KUKA KRL program: MyProgram_267().src

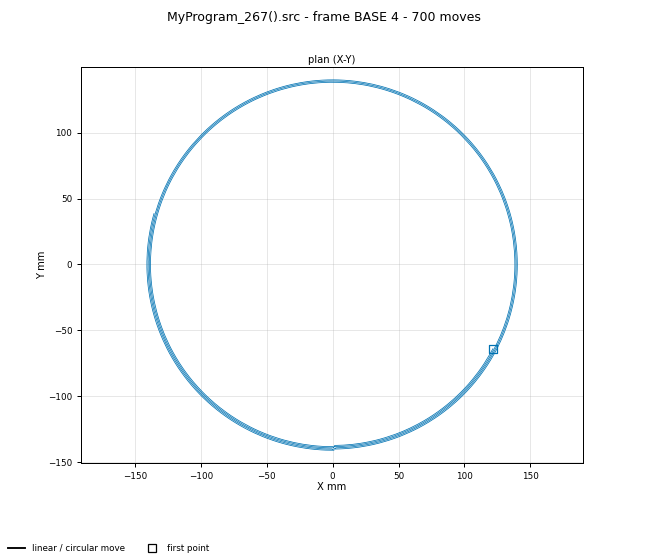
[picture p0: tool path of MyProgram_267().src in frame BASE 4, 700 of 700 moves have a stored position in this frame; points joined in program order, loops and branches not executed]
&ACCESS RVP
&REL 1
&PARAM TEMPLATE = C:\KRC\Roboter\Template\vorgabe
&PARAM EDITMASK = *
DEF MyProgram_267()
; ---- Setting reference (Base) ----
$BASE = BASE_DATA[4]

; --------------------------
; ---- Setting tool (TCP) ----
$TOOL = TOOL_DATA[3]
; --------------------------

$VEL.CP = VEL_APROX_PRINT
Startdeposition()
$VEL.CP = VEL_PRINT
LIN {X 121.5223,Y -63.9531,Z 169,A -26.4132,B 9.7444,C 0.283,E1 9.8897,E2 477.634} C_DIS
LIN {X 119.4927,Y -67.6748,Z 169,A -28.3857,B 9.744,C 0.2925,E1 9.8869,E2 479.6342} C_DIS
LIN {X 114.8477,Y -75.2879,Z 169,A -31.797,B 9.744,C 0.2945,E1 9.882,E2 483.0104} C_DIS
LIN {X 112.9327,Y -78.1315,Z 169,A -33.3387,B 9.7438,C 0.3007,E1 9.8795,E2 484.5678} C_DIS
LIN {X 110.5893,Y -81.4139,Z 169,A -34.9698,B 9.7438,C 0.3035,E1 9.8769,E2 486.1941} C_DIS
LIN {X 107.7784,Y -85.1007,Z 169,A -36.6917,B 9.7438,C 0.303,E1 9.874,E2 487.8912} C_DIS
LIN {X 105.9489,Y -87.3676,Z 169,A -38.1579,B 9.7434,C 0.3119,E1 9.8713,E2 489.3904} C_DIS
LIN {X 103.0991,Y -90.7131,Z 169,A -40.1493,B 9.7432,C 0.3198,E1 9.8676,E2 491.4037} C_DIS
LIN {X 100.8727,Y -93.1825,Z 169,A -41.7921,B 9.7429,C 0.3289,E1 9.8645,E2 493.08} C_DIS
LIN {X 97.5521,Y -96.653,Z 169,A -43.3158,B 9.7431,C 0.3219,E1 9.8616,E2 494.5453} C_DIS
LIN {X 92.7016,Y -101.3149,Z 169,A -46.0443,B 9.743,C 0.3259,E1 9.8561,E2 497.2667} C_DIS
LIN {X 87.8927,Y -105.5141,Z 169,A -48.4523,B 9.743,C 0.3252,E1 9.8511,E2 499.6449} C_DIS
LIN {X 83.878,Y -108.7326,Z 169,A -51.2584,B 9.7423,C 0.3447,E1 9.8447,E2 502.5365} C_DIS
LIN {X 80.2624,Y -111.4281,Z 169,A -52.6799,B 9.7426,C 0.3374,E1 9.8416,E2 503.9017} C_DIS
LIN {X 76.6421,Y -113.9489,Z 169,A -54.4958,B 9.7426,C 0.34,E1 9.8374,E2 505.7163} C_DIS
LIN {X 73.1697,Y -116.2085,Z 169,A -56.1855,B 9.7424,C 0.342,E1 9.8335,E2 507.4026} C_DIS
LIN {X 69.7328,Y -118.3029,Z 169,A -57.7924,B 9.7424,C 0.343,E1 9.8296,E2 509.0019} C_DIS
LIN {X 64.6366,Y -121.163,Z 169,A -60.2336,B 9.7423,C 0.3468,E1 9.8237,E2 511.4457} C_DIS
LIN {X 61.9846,Y -122.5384,Z 169,A -61.5098,B 9.7422,C 0.3493,E1 9.8205,E2 512.7266} C_DIS
LIN {X 58.8364,Y -124.081,Z 169,A -62.8714,B 9.7422,C 0.349,E1 9.8171,E2 514.0767} C_DIS
LIN {X 54.0796,Y -126.227,Z 169,A -65.0052,B 9.7422,C 0.3508,E1 9.8117,E2 516.2068} C_DIS
LIN {X 51.4311,Y -127.3284,Z 169,A -66.2612,B 9.742,C 0.3536,E1 9.8084,E2 517.4712} C_DIS
LIN {X 47.3484,Y -128.9049,Z 169,A -68.3007,B 9.7418,C 0.3606,E1 9.803,E2 519.5393} C_DIS
LIN {X 42.0304,Y -130.7333,Z 169,A -70.1991,B 9.7421,C 0.3529,E1 9.7981,E2 521.3826} C_DIS
LIN {X 40.0355,Y -131.3578,Z 169,A -71.2939,B 9.7418,C 0.3588,E1 9.7951,E2 522.5064} C_DIS
LIN {X 36.2701,Y -132.449,Z 169,A -72.8975,B 9.7418,C 0.3596,E1 9.7908,E2 524.1071} C_DIS
LIN {X 32.8798,Y -133.331,Z 169,A -74.3211,B 9.7418,C 0.3599,E1 9.787,E2 525.5269} C_DIS
LIN {X 28.4405,Y -134.3472,Z 169,A -76.2879,B 9.7417,C 0.3629,E1 9.7816,E2 527.5034} C_DIS
LIN {X 25.1446,Y -135.0034,Z 169,A -77.8597,B 9.7415,C 0.3675,E1 9.7772,E2 529.0976} C_DIS
LIN {X 21.1222,Y -135.6894,Z 169,A -79.3371,B 9.7417,C 0.3636,E1 9.7732,E2 530.5475} C_DIS
LIN {X 15.2674,Y -136.4735,Z 169,A -81.7848,B 9.7417,C 0.3645,E1 9.7664,E2 532.9947} C_DIS
LIN {X 8.3393,Y -137.0702,Z 169,A -84.7346,B 9.7416,C 0.3666,E1 9.7582,E2 535.9522} C_DIS
LIN {X 1.6144,Y -137.3159,Z 169,A -87.597,B 9.7415,C 0.3684,E1 9.7502,E2 538.8231} C_DIS
LIN {X 1.6144,Y -137.3159,Z 169,A -87.597,B 9.7415,C 0.3684,E1 9.7502,E2 538.8231} C_DIS
Enddeposition()
LIN {X 1.0035,Y -138.2302,Z 169,A -87.3337,B 9.7081,C 0.3639,E1 9.7175,E2 538.5378} C_DIS
Startdeposition()
$VEL.CP = VEL_PRINT
LIN {X 3.6243,Y -138.1887,Z 169,A -85.9275,B 9.7084,C 0.3567,E1 9.7215,E2 537.0898} C_DIS
LIN {X 8.1585,Y -137.9955,Z 169,A -84.3267,B 9.7082,C 0.3624,E1 9.7259,E2 535.5242} C_DIS
LIN {X 12.5987,Y -137.662,Z 169,A -82.2235,B 9.7084,C 0.3561,E1 9.7318,E2 533.3868} C_DIS
LIN {X 15.47,Y -137.3693,Z 169,A -80.2721,B 9.709,C 0.3386,E1 9.7375,E2 531.3363} C_DIS
LIN {X 21.6232,Y -136.5351,Z 169,A -78.7263,B 9.7082,C 0.3603,E1 9.7414,E2 529.9229} C_DIS
LIN {X 27.0044,Y -135.5737,Z 169,A -76.2156,B 9.7085,C 0.3533,E1 9.7484,E2 527.3791} C_DIS
LIN {X 31.4408,Y -134.6145,Z 169,A -73.9888,B 9.7088,C 0.344,E1 9.7546,E2 525.1061} C_DIS
LIN {X 35.2299,Y -133.6717,Z 169,A -72.753,B 9.7086,C 0.3514,E1 9.7578,E2 523.9189} C_DIS
LIN {X 38.6757,Y -132.7152,Z 169,A -71.3127,B 9.7086,C 0.351,E1 9.7616,E2 522.483} C_DIS
LIN {X 42.1668,Y -131.6475,Z 169,A -69.2693,B 9.7091,C 0.3373,E1 9.7673,E2 520.3694} C_DIS
LIN {X 46.617,Y -130.1385,Z 169,A -68.083,B 9.7085,C 0.3527,E1 9.7702,E2 519.2806} C_DIS
LIN {X 51.6048,Y -128.2421,Z 169,A -65.7308,B 9.7087,C 0.3469,E1 9.7763,E2 516.9086} C_DIS
LIN {X 58.3851,Y -125.3013,Z 169,A -62.6142,B 9.7089,C 0.3418,E1 9.7843,E2 513.7827} C_DIS
LIN {X 62.2786,Y -123.4126,Z 169,A -60.8218,B 9.7089,C 0.3393,E1 9.7888,E2 511.989} C_DIS
LIN {X 65.0912,Y -121.9545,Z 169,A -59.5881,B 9.7089,C 0.3393,E1 9.7918,E2 510.7645} C_DIS
LIN {X 68.9115,Y -119.8373,Z 169,A -57.5572,B 9.7093,C 0.3313,E1 9.7968,E2 508.7033} C_DIS
LIN {X 73.8951,Y -116.8295,Z 169,A -55.2807,B 9.7093,C 0.3305,E1 9.8022,E2 506.4423} C_DIS
LIN {X 77.7185,Y -114.322,Z 169,A -53.6415,B 9.7092,C 0.3333,E1 9.8059,E2 504.8345} C_DIS
LIN {X 81.5319,Y -111.6347,Z 169,A -50.4812,B 9.7103,C 0.3005,E1 9.8135,E2 501.5122} C_DIS
LIN {X 87.6058,Y -106.9339,Z 169,A -47.584,B 9.7103,C 0.3013,E1 9.8196,E2 498.6497} C_DIS
LIN {X 92.3827,Y -102.8352,Z 169,A -45.9634,B 9.7096,C 0.3198,E1 9.8228,E2 497.1552} C_DIS
LIN {X 96.5302,Y -98.9528,Z 169,A -43.3774,B 9.71,C 0.3094,E1 9.8281,E2 494.537} C_DIS
LIN {X 102.34,Y -92.9307,Z 169,A -40.2491,B 9.71,C 0.31,E1 9.834,E2 491.4493} C_DIS
LIN {X 105.7678,Y -89.0102,Z 169,A -37.829,B 9.7103,C 0.2988,E1 9.8385,E2 488.9932} C_DIS
LIN {X 110.706,Y -82.7881,Z 169,A -34.445,B 9.7106,C 0.2888,E1 9.8443,E2 485.5939} C_DIS
LIN {X 113.6513,Y -78.6962,Z 169,A -32.5038,B 9.7106,C 0.2873,E1 9.8474,E2 483.6697} C_DIS
LIN {X 115.518,Y -75.929,Z 169,A -30.804,B 9.711,C 0.2761,E1 9.8501,E2 481.9274} C_DIS
LIN {X 117.7858,Y -72.361,Z 169,A -29.4472,B 9.7108,C 0.2813,E1 9.852,E2 480.62} C_DIS
LIN {X 119.8827,Y -68.8324,Z 169,A -27.7305,B 9.711,C 0.2766,E1 9.8544,E2 478.8995} C_DIS
LIN {X 121.9811,Y -65.0416,Z 169,A -25.9549,B 9.711,C 0.2724,E1 9.8568,E2 477.1247} C_DIS
LIN {X 124.1565,Y -60.7815,Z 169,A -23.1233,B 9.7118,C 0.2461,E1 9.8604,E2 474.1803} C_DIS
LIN {X 127.1987,Y -54.1312,Z 169,A -21.0317,B 9.7114,C 0.2612,E1 9.8626,E2 472.2079} C_DIS
LIN {X 129.7662,Y -47.6495,Z 169,A -18.1375,B 9.7116,C 0.2531,E1 9.8655,E2 469.3101} C_DIS
LIN {X 131.1674,Y -43.6372,Z 169,A -16.5544,B 9.7116,C 0.2526,E1 9.8669,E2 467.748} C_DIS
LIN {X 132.0304,Y -40.9555,Z 169,A -14.6508,B 9.7121,C 0.2311,E1 9.8686,E2 465.7479} C_DIS
LIN {X 133.6372,Y -35.3594,Z 169,A -12.9817,B 9.7119,C 0.2427,E1 9.8697,E2 464.1727} C_DIS
LIN {X 134.6403,Y -31.3276,Z 169,A -11.2449,B 9.7119,C 0.2374,E1 9.8709,E2 462.4322} C_DIS
LIN {X 136.0297,Y -24.5995,Z 169,A -8.547,B 9.7121,C 0.2329,E1 9.8723,E2 459.7506} C_DIS
LIN {X 137.2624,Y -16.3765,Z 169,A -5.3848,B 9.7121,C 0.23,E1 9.8736,E2 456.6214} C_DIS
LIN {X 137.5318,Y -13.94,Z 169,A -3.6442,B 9.7126,C 0.2091,E1 9.8741,E2 454.7869} C_DIS
LIN {X 137.9056,Y -9.5653,Z 169,A -2.3869,B 9.7124,C 0.2178,E1 9.8744,E2 453.6001} C_DIS
LIN {X 138.1517,Y -4.8579,Z 169,A -0.3244,B 9.7126,C 0.2094,E1 9.8746,E2 451.5217} C_DIS
LIN {X 138.2326,Y -1.1208,Z 169,A 1.7321,B 9.713,C 0.1923,E1 9.8746,E2 449.3985} C_DIS
LIN {X 138.1805,Y 3.9204,Z 169,A 3.8684,B 9.7131,C 0.185,E1 9.8745,E2 447.2541} C_DIS
LIN {X 137.9104,Y 9.4997,Z 169,A 5.533,B 9.7129,C 0.1944,E1 9.8742,E2 445.6712} C_DIS
LIN {X 137.1413,Y 17.3717,Z 169,A 8.5943,B 9.713,C 0.1903,E1 9.8733,E2 442.6347} C_DIS
LIN {X 136.3718,Y 22.6254,Z 169,A 10.9146,B 9.7132,C 0.1811,E1 9.8723,E2 440.2971} C_DIS
LIN {X 135.6149,Y 26.8018,Z 169,A 12.8909,B 9.7134,C 0.1707,E1 9.8713,E2 438.2917} C_DIS
LIN {X 134.9256,Y 30.0788,Z 169,A 14.0849,B 9.7134,C 0.1716,E1 9.8706,E2 437.1213} C_DIS
LIN {X 134.0282,Y 33.8467,Z 169,A 15.5369,B 9.7134,C 0.1708,E1 9.8696,E2 435.6875} C_DIS
LIN {X 133.1585,Y 37.1205,Z 169,A 16.9008,B 9.7134,C 0.1678,E1 9.8686,E2 434.3275} C_DIS
LIN {X 132.2106,Y 40.3666,Z 169,A 18.3307,B 9.7135,C 0.1632,E1 9.8675,E2 432.8929} C_DIS
LIN {X 131.1435,Y 43.7089,Z 169,A 19.7573,B 9.7135,C 0.1599,E1 9.8662,E2 431.4687} C_DIS
LIN {X 130.0245,Y 46.933,Z 169,A 21.422,B 9.7137,C 0.15,E1 9.8646,E2 429.771} C_DIS
LIN {X 128.8641,Y 50.0313,Z 169,A 22.6119,B 9.7137,C 0.1507,E1 9.8635,E2 428.6033} C_DIS
LIN {X 127.1009,Y 54.3573,Z 169,A 24.3261,B 9.7137,C 0.1509,E1 9.8617,E2 426.9159} C_DIS
LIN {X 125.6911,Y 57.5421,Z 169,A 25.6983,B 9.7137,C 0.1488,E1 9.8601,E2 425.5518} C_DIS
LIN {X 124.288,Y 60.5148,Z 169,A 27.2672,B 9.7139,C 0.1403,E1 9.8582,E2 423.9559} C_DIS
LIN {X 122.5937,Y 63.875,Z 169,A 28.7368,B 9.7139,C 0.1385,E1 9.8563,E2 422.4966} C_DIS
LIN {X 120.4568,Y 67.8217,Z 169,A 30.5977,B 9.7139,C 0.1338,E1 9.8538,E2 420.6345} C_DIS
LIN {X 117.4731,Y 72.8679,Z 169,A 33.0483,B 9.714,C 0.1273,E1 9.8503,E2 418.1799} C_DIS
LIN {X 115.0774,Y 76.5952,Z 169,A 34.8875,B 9.714,C 0.1228,E1 9.8474,E2 416.3394} C_DIS
LIN {X 112.2801,Y 80.6403,Z 169,A 36.8588,B 9.7141,C 0.1196,E1 9.8443,E2 414.3755} C_DIS
LIN {X 110.4497,Y 83.1294,Z 169,A 38.5654,B 9.7143,C 0.1065,E1 9.8413,E2 412.6141} C_DIS
LIN {X 107.5833,Y 86.8069,Z 169,A 40.1356,B 9.7143,C 0.1108,E1 9.8387,E2 411.0891} C_DIS
LIN {X 104.4049,Y 90.6056,Z 169,A 41.928,B 9.7143,C 0.1125,E1 9.8355,E2 409.3287} C_DIS
LIN {X 97.6535,Y 97.8442,Z 169,A 45.8298,B 9.7143,C 0.1087,E1 9.8281,E2 405.451} C_DIS
LIN {X 94.3854,Y 101.0003,Z 169,A 48.007,B 9.7143,C 0.0981,E1 9.8236,E2 403.2363} C_DIS
LIN {X 91.0289,Y 104.0355,Z 169,A 49.7708,B 9.7143,C 0.0971,E1 9.8199,E2 401.486} C_DIS
LIN {X 86.2559,Y 108.0258,Z 169,A 52.43,B 9.7144,C 0.0906,E1 9.8142,E2 398.816} C_DIS
LIN {X 82.0554,Y 111.2501,Z 169,A 55.1586,B 9.7146,C 0.0744,E1 9.8079,E2 396.0195} C_DIS
LIN {X 77.6146,Y 114.3924,Z 169,A 56.808,B 9.7145,C 0.0848,E1 9.8043,E2 394.4463} C_DIS
LIN {X 73.7755,Y 116.905,Z 169,A 58.6399,B 9.7145,C 0.0834,E1 9.8,E2 392.6229} C_DIS
LIN {X 70.2078,Y 119.082,Z 169,A 60.4141,B 9.7145,C 0.0799,E1 9.7957,E2 390.8433} C_DIS
LIN {X 66.413,Y 121.2394,Z 169,A 62.1811,B 9.7145,C 0.0784,E1 9.7914,E2 389.0814} C_DIS
LIN {X 58.9104,Y 125.0567,Z 169,A 65.5976,B 9.7145,C 0.0756,E1 9.7829,E2 385.6741} C_DIS
LIN {X 55.2301,Y 126.7236,Z 169,A 67.2877,B 9.7145,C 0.0733,E1 9.7786,E2 383.982} C_DIS
LIN {X 50.5322,Y 128.6694,Z 169,A 69.4095,B 9.7146,C 0.0708,E1 9.7731,E2 381.8586} C_DIS
LIN {X 47.1906,Y 129.9316,Z 169,A 70.8642,B 9.7146,C 0.0699,E1 9.7693,E2 380.4073} C_DIS
LIN {X 43.8069,Y 131.1109,Z 169,A 72.2508,B 9.7146,C 0.0707,E1 9.7657,E2 379.0331} C_DIS
LIN {X 40.5239,Y 132.1625,Z 169,A 73.7076,B 9.7146,C 0.0689,E1 9.7618,E2 377.5731} C_DIS
LIN {X 37.2525,Y 133.1216,Z 169,A 75.1127,B 9.7146,C 0.068,E1 9.758,E2 376.1693} C_DIS
LIN {X 33.8959,Y 134.0157,Z 169,A 77.457,B 9.7147,C 0.0472,E1 9.7514,E2 373.7115} C_DIS
LIN {X 27.4409,Y 135.4849,Z 169,A 79.3116,B 9.7147,C 0.0651,E1 9.7466,E2 371.9696} C_DIS
LIN {X 23.3469,Y 136.2514,Z 169,A 80.9226,B 9.7147,C 0.0667,E1 9.7422,E2 370.3735} C_DIS
LIN {X 16.9282,Y 137.1966,Z 169,A 83.5898,B 9.7147,C 0.0662,E1 9.7349,E2 367.7099} C_DIS
LIN {X 11.2415,Y 137.7787,Z 169,A 86.0643,B 9.7147,C 0.0634,E1 9.7279,E2 365.2233} C_DIS
LIN {X 4.1252,Y 138.1748,Z 169,A 89.0412,B 9.7147,C 0.0626,E1 9.7196,E2 362.2449} C_DIS
LIN {X -1.4773,Y 138.2301,Z 169,A 91.4614,B 9.7147,C 0.0606,E1 9.7128,E2 359.8137} C_DIS
LIN {X -4.6109,Y 138.1612,Z 169,A 93.452,B 9.7147,C 0.0462,E1 9.7071,E2 357.7371} C_DIS
LIN {X -10.677,Y 137.8244,Z 169,A 95.3517,B 9.7147,C 0.0598,E1 9.702,E2 355.9164} C_DIS
LIN {X -15.8973,Y 137.3196,Z 169,A 97.4052,B 9.7147,C 0.0631,E1 9.6963,E2 353.879} C_DIS
LIN {X -18.8245,Y 136.9502,Z 169,A 99.1396,B 9.7147,C 0.053,E1 9.6914,E2 352.0815} C_DIS
LIN {X -23.5939,Y 136.2096,Z 169,A 100.6893,B 9.7147,C 0.0634,E1 9.6872,E2 350.5895} C_DIS
LIN {X -28.7916,Y 135.2048,Z 169,A 102.7072,B 9.7147,C 0.0683,E1 9.6818,E2 348.5948} C_DIS
LIN {X -31.8808,Y 134.5103,Z 169,A 104.1791,B 9.7147,C 0.0659,E1 9.6777,E2 347.104} C_DIS
LIN {X -35.5184,Y 133.5948,Z 169,A 105.5905,B 9.7147,C 0.07,E1 9.6739,E2 345.7115} C_DIS
LIN {X -38.5661,Y 132.7473,Z 169,A 106.9576,B 9.7147,C 0.07,E1 9.6703,E2 344.3383} C_DIS
LIN {X -41.9093,Y 131.7298,Z 169,A 108.392,B 9.7147,C 0.0716,E1 9.6664,E2 342.9067} C_DIS
LIN {X -47.9387,Y 129.6579,Z 169,A 111.2253,B 9.7147,C 0.0704,E1 9.6589,E2 340.0518} C_DIS
LIN {X -51.8181,Y 128.1561,Z 169,A 112.7433,B 9.7146,C 0.0764,E1 9.655,E2 338.5607} C_DIS
LIN {X -54.9202,Y 126.8576,Z 169,A 114.1713,B 9.7146,C 0.0773,E1 9.6514,E2 337.1295} C_DIS
LIN {X -57.7435,Y 125.5979,Z 169,A 115.5007,B 9.7146,C 0.078,E1 9.648,E2 335.7953} C_DIS
LIN {X -60.1655,Y 124.4571,Z 169,A 116.7467,B 9.7146,C 0.0768,E1 9.6448,E2 334.5333} C_DIS
LIN {X -63.9261,Y 122.5669,Z 169,A 118.3999,B 9.7146,C 0.0809,E1 9.6407,E2 332.8928} C_DIS
LIN {X -66.7962,Y 121.0286,Z 169,A 120.3317,B 9.7146,C 0.0715,E1 9.6358,E2 330.8897} C_DIS
LIN {X -71.0467,Y 118.5836,Z 169,A 121.9053,B 9.7146,C 0.0835,E1 9.6322,E2 329.3753} C_DIS
LIN {X -75.4987,Y 115.8,Z 169,A 124.0805,B 9.7145,C 0.087,E1 9.6271,E2 327.2021} C_DIS
LIN {X -79.2712,Y 113.2508,Z 169,A 126.1506,B 9.7145,C 0.0867,E1 9.6223,E2 325.111} C_DIS
LIN {X -83.8964,Y 109.8681,Z 169,A 128.455,B 9.7145,C 0.0922,E1 9.6171,E2 322.8176} C_DIS
LIN {X -87.7527,Y 106.8138,Z 169,A 130.4515,B 9.7144,C 0.0969,E1 9.6128,E2 320.8284} C_DIS
LIN {X -91.1352,Y 103.9427,Z 169,A 132.215,B 9.7144,C 0.1018,E1 9.6091,E2 319.0761} C_DIS
LIN {X -93.5689,Y 101.7569,Z 169,A 133.9184,B 9.7144,C 0.098,E1 9.6055,E2 317.3307} C_DIS
LIN {X -96.1599,Y 99.312,Z 169,A 135.1329,B 9.7143,C 0.106,E1 9.6031,E2 316.1503} C_DIS
LIN {X -99.2052,Y 96.2702,Z 169,A 136.9867,B 9.7143,C 0.1084,E1 9.5995,E2 314.2897} C_DIS
LIN {X -104.0773,Y 90.981,Z 169,A 139.9896,B 9.7142,C 0.1145,E1 9.5939,E2 311.2871} C_DIS
LIN {X -107.0454,Y 87.4693,Z 169,A 141.8221,B 9.7142,C 0.1202,E1 9.5906,E2 309.4657} C_DIS
LIN {X -109.4058,Y 84.498,Z 169,A 143.6667,B 9.7142,C 0.1188,E1 9.5874,E2 307.5888} C_DIS
LIN {X -112.6331,Y 80.1467,Z 169,A 145.8081,B 9.7141,C 0.1261,E1 9.5839,E2 305.4628} C_DIS
LIN {X -115.1812,Y 76.4398,Z 169,A 147.5419,B 9.714,C 0.1331,E1 9.5812,E2 303.7473} C_DIS
LIN {X -117.7625,Y 72.399,Z 169,A 149.4895,B 9.7139,C 0.1388,E1 9.5783,E2 301.8068} C_DIS
LIN {X -121.4641,Y 66.0011,Z 169,A 152.7744,B 9.7139,C 0.1426,E1 9.5738,E2 298.4977} C_DIS
LIN {X -123.106,Y 62.8809,Z 169,A 154.13,B 9.7137,C 0.1483,E1 9.572,E2 297.1568} C_DIS
LIN {X -124.8544,Y 59.334,Z 169,A 155.8728,B 9.7137,C 0.1507,E1 9.5699,E2 295.4028} C_DIS
LIN {X -126.5527,Y 55.6253,Z 169,A 157.691,B 9.7137,C 0.153,E1 9.5678,E2 293.5705} C_DIS
LIN {X -128.077,Y 52.0142,Z 169,A 159.1678,B 9.7136,C 0.1601,E1 9.5662,E2 292.1139} C_DIS
LIN {X -129.2518,Y 49.0241,Z 169,A 160.8875,B 9.7136,C 0.1566,E1 9.5645,E2 290.3471} C_DIS
LIN {X -130.4518,Y 45.7344,Z 169,A 162.0752,B 9.7135,C 0.1655,E1 9.5634,E2 289.194} C_DIS
LIN {X -131.5709,Y 42.4066,Z 169,A 163.4888,B 9.7134,C 0.1703,E1 9.5622,E2 287.7872} C_DIS
LIN {X -132.6389,Y 38.9365,Z 169,A 165.0911,B 9.7134,C 0.1727,E1 9.5609,E2 286.1742} C_DIS
LIN {X -133.7242,Y 35.0331,Z 169,A 166.8197,B 9.7133,C 0.1766,E1 9.5596,E2 284.4412} C_DIS
LIN {X -134.6959,Y 31.0843,Z 169,A 168.5005,B 9.7132,C 0.1815,E1 9.5586,E2 282.7627} C_DIS
LIN {X -135.4504,Y 27.6101,Z 169,A 169.9415,B 9.7131,C 0.1863,E1 9.5577,E2 281.3273} C_DIS
LIN {X -136.0924,Y 24.2491,Z 169,A 171.4124,B 9.7131,C 0.1894,E1 9.557,E2 279.8513} C_DIS
LIN {X -136.7404,Y 20.2923,Z 169,A 173.1172,B 9.713,C 0.1934,E1 9.5563,E2 278.1429} C_DIS
LIN {X -137.255,Y 16.4394,Z 169,A 174.7144,B 9.7129,C 0.1984,E1 9.5557,E2 276.5491} C_DIS
LIN {X -137.8186,Y 10.7537,Z 169,A 177.3369,B 9.7129,C 0.2006,E1 9.555,E2 273.897} C_DIS
LIN {X -138.1191,Y 5.6939,Z 169,A 179.2691,B 9.7126,C 0.2098,E1 9.5548,E2 271.9881} C_DIS
LIN {X -138.2299,Y 1.4816,Z 169,A -178.6784,B 9.7126,C 0.2093,E1 9.5547,E2 269.8987} C_DIS
LIN {X -138.2253,Y -1.7932,Z 169,A -177.3012,B 9.7126,C 0.2129,E1 9.5547,E2 268.5203} C_DIS
LIN {X -138.1426,Y -5.0909,Z 169,A -176.2193,B 9.7123,C 0.2221,E1 9.5548,E2 267.4758} C_DIS
LIN {X -137.9596,Y -8.7402,Z 169,A -174.6605,B 9.7123,C 0.2257,E1 9.5551,E2 265.9128} C_DIS
LIN {X -137.7049,Y -12.1148,Z 169,A -173.0647,B 9.7123,C 0.2262,E1 9.5554,E2 264.2939} C_DIS
LIN {X -137.2252,Y -16.6889,Z 169,A -171.2799,B 9.7121,C 0.234,E1 9.556,E2 262.5261} C_DIS
LIN {X -136.6572,Y -20.8342,Z 169,A -169.5285,B 9.712,C 0.2386,E1 9.5567,E2 260.7741} C_DIS
LIN {X -136.0705,Y -24.3715,Z 169,A -167.9831,B 9.7119,C 0.2418,E1 9.5574,E2 259.2225} C_DIS
LIN {X -135.1822,Y -28.8959,Z 169,A -166.0957,B 9.7117,C 0.2476,E1 9.5585,E2 257.3397} C_DIS
LIN {X -134.4286,Y -32.2198,Z 169,A -164.6815,B 9.7117,C 0.2516,E1 9.5594,E2 255.9265} C_DIS
LIN {X -133.6216,Y -35.418,Z 169,A -163.3442,B 9.7115,C 0.256,E1 9.5603,E2 254.5941} C_DIS
LIN {X -132.4499,Y -39.5786,Z 169,A -161.1531,B 9.7115,C 0.2536,E1 9.5621,E2 252.3538} C_DIS
LIN {X -131.4087,Y -42.9125,Z 169,A -159.8914,B 9.7114,C 0.261,E1 9.5631,E2 251.117} C_DIS
LIN {X -129.9324,Y -47.1887,Z 169,A -158.0159,B 9.7113,C 0.2661,E1 9.5649,E2 249.2428} C_DIS
LIN {X -128.3876,Y -51.2437,Z 169,A -156.3394,B 9.7111,C 0.2731,E1 9.5666,E2 247.5831} C_DIS
LIN {X -127.0594,Y -54.4533,Z 169,A -154.8143,B 9.711,C 0.2754,E1 9.5682,E2 246.0481} C_DIS
LIN {X -125.4828,Y -57.9925,Z 169,A -153.2096,B 9.7109,C 0.2796,E1 9.5701,E2 244.4447} C_DIS
LIN {X -124.1254,Y -60.8444,Z 169,A -151.8593,B 9.7109,C 0.2822,E1 9.5717,E2 243.0901} C_DIS
LIN {X -122.7213,Y -63.6321,Z 169,A -150.1834,B 9.7109,C 0.2783,E1 9.5739,E2 241.3664} C_DIS
LIN {X -120.9828,Y -66.8788,Z 169,A -148.9717,B 9.7106,C 0.2881,E1 9.5755,E2 240.1957} C_DIS
LIN {X -118.8307,Y -70.6322,Z 169,A -147.0917,B 9.7106,C 0.2909,E1 9.5782,E2 238.3059} C_DIS
LIN {X -116.5476,Y -74.3392,Z 169,A -145.2667,B 9.7104,C 0.2948,E1 9.5809,E2 236.4792} C_DIS
LIN {X -114.119,Y -78.0162,Z 169,A -143.384,B 9.7104,C 0.2981,E1 9.5838,E2 234.5903} C_DIS
LIN {X -112.0041,Y -81.0228,Z 169,A -141.775,B 9.7103,C 0.3,E1 9.5865,E2 232.9712} C_DIS
LIN {X -109.0102,Y -85.0091,Z 169,A -139.7469,B 9.7101,C 0.3053,E1 9.5899,E2 230.9491} C_DIS
LIN {X -106.1549,Y -88.5489,Z 169,A -138.1373,B 9.7098,C 0.3147,E1 9.5927,E2 229.3755} C_DIS
LIN {X -102.0651,Y -93.2336,Z 169,A -135.2706,B 9.7098,C 0.3147,E1 9.5981,E2 226.4731} C_DIS
LIN {X -99.0785,Y -96.401,Z 169,A -133.5754,B 9.7096,C 0.3204,E1 9.6013,E2 224.7925} C_DIS
LIN {X -96.4308,Y -99.0498,Z 169,A -131.8388,B 9.7096,C 0.3199,E1 9.6048,E2 223.0328} C_DIS
LIN {X -93.1033,Y -102.1834,Z 169,A -130.0244,B 9.7095,C 0.3251,E1 9.6085,E2 221.2293} C_DIS
LIN {X -89.3665,Y -105.467,Z 169,A -127.8921,B 9.7094,C 0.3274,E1 9.613,E2 219.0886} C_DIS
LIN {X -85.8593,Y -108.3414,Z 169,A -125.986,B 9.7094,C 0.3302,E1 9.6171,E2 217.1795} C_DIS
LIN {X -80.6381,Y -112.2817,Z 169,A -123.2098,B 9.7092,C 0.3333,E1 9.6234,E2 214.3955} C_DIS
LIN {X -76.9859,Y -114.8166,Z 169,A -121.5379,B 9.709,C 0.3396,E1 9.6272,E2 212.7459} C_DIS
LIN {X -73.3704,Y -117.1603,Z 169,A -119.5483,B 9.709,C 0.3381,E1 9.6319,E2 210.7303} C_DIS
LIN {X -69.4751,Y -119.511,Z 169,A -117.6716,B 9.709,C 0.3409,E1 9.6365,E2 208.8549} C_DIS
LIN {X -62.4196,Y -123.3408,Z 169,A -114.384,B 9.7088,C 0.346,E1 9.6446,E2 205.5727} C_DIS
LIN {X -58.8512,Y -125.085,Z 169,A -112.7425,B 9.7087,C 0.348,E1 9.6487,E2 203.9319} C_DIS
LIN {X -55.2614,Y -126.71,Z 169,A -110.9933,B 9.7087,C 0.3473,E1 9.6532,E2 202.1676} C_DIS
LIN {X -51.3412,Y -128.3483,Z 169,A -109.3294,B 9.7086,C 0.3511,E1 9.6574,E2 200.5161} C_DIS
LIN {X -47.2274,Y -129.9184,Z 169,A -107.502,B 9.7086,C 0.3527,E1 9.6622,E2 198.6882} C_DIS
LIN {X -44.0678,Y -131.024,Z 169,A -106.1927,B 9.7084,C 0.3554,E1 9.6657,E2 197.3887} C_DIS
LIN {X -40.8384,Y -132.0662,Z 169,A -104.6958,B 9.7084,C 0.3546,E1 9.6697,E2 195.8801} C_DIS
LIN {X -36.5726,Y -133.3117,Z 169,A -101.8235,B 9.7092,C 0.334,E1 9.6778,E2 192.8733} C_DIS
LIN {X -29.4181,Y -135.0695,Z 169,A -99.7751,B 9.7084,C 0.3571,E1 9.683,E2 190.9552} C_DIS
LIN {X -25.8933,Y -135.7891,Z 169,A -98.0348,B 9.7085,C 0.3524,E1 9.6879,E2 189.1822} C_DIS
LIN {X -22.697,Y -136.3598,Z 169,A -96.8183,B 9.7085,C 0.3557,E1 9.6912,E2 187.982} C_DIS
LIN {X -15.6225,Y -137.3521,Z 169,A -93.8885,B 9.7084,C 0.3571,E1 9.6993,E2 185.0554} C_DIS
LIN {X -11.897,Y -137.7233,Z 169,A -92.3052,B 9.7084,C 0.3566,E1 9.7037,E2 183.4674} C_DIS
LIN {X -7.36,Y -138.0406,Z 169,A -90.6024,B 9.7082,C 0.3607,E1 9.7084,E2 181.7875} C_DIS
LIN {X -3.7361,Y -138.1856,Z 169,A -89.0514,B 9.7082,C 0.3596,E1 9.7127,E2 180.2296} C_DIS
LIN {X 0.268,Y -138.2368,Z 169,A -87.3639,B 9.7082,C 0.3588,E1 9.7174,E2 178.5378} C_DIS
LIN {X 0.268,Y -138.2368,Z 169,A -87.3639,B 9.7082,C 0.3588,E1 9.7174,E2 178.5378} C_DIS
Enddeposition()
LIN {X 1.014,Y -139.143,Z 169,A -87.126,B 9.5898,C 0.3694,E1 9.5998,E2 178.3775} C_DIS
Startdeposition()
$VEL.CP = VEL_PRINT
LIN {X -2.5474,Y -139.1253,Z 169,A -89.1002,B 9.5893,C 0.3805,E1 9.5941,E2 180.4183} C_DIS
LIN {X -6.4133,Y -139.0017,Z 169,A -90.8085,B 9.5893,C 0.383,E1 9.5893,E2 182.1422} C_DIS
LIN {X -11.3884,Y -138.6819,Z 169,A -92.8192,B 9.5893,C 0.382,E1 9.5837,E2 184.1483} C_DIS
LIN {X -15.3156,Y -138.3035,Z 169,A -94.4156,B 9.5893,C 0.3811,E1 9.5793,E2 185.7417} C_DIS
LIN {X -20.2715,Y -137.665,Z 169,A -96.4893,B 9.5893,C 0.3809,E1 9.5736,E2 187.8182} C_DIS
LIN {X -27.1692,Y -136.4712,Z 169,A -100.608,B 9.5883,C 0.4052,E1 9.5618,E2 192.0949} C_DIS
LIN {X -35.5577,Y -134.5285,Z 169,A -103.012,B 9.5894,C 0.3797,E1 9.5557,E2 194.3548} C_DIS
LIN {X -39.6517,Y -133.3801,Z 169,A -104.6288,B 9.5895,C 0.3758,E1 9.5514,E2 195.9547} C_DIS
LIN {X -42.5502,Y -132.4828,Z 169,A -105.8966,B 9.5895,C 0.3752,E1 9.548,E2 197.2251} C_DIS
LIN {X -45.8609,Y -131.3736,Z 169,A -107.3454,B 9.5895,C 0.3742,E1 9.5442,E2 198.6755} C_DIS
LIN {X -49.118,Y -130.191,Z 169,A -108.7942,B 9.5896,C 0.3734,E1 9.5404,E2 200.1273} C_DIS
LIN {X -52.2095,Y -128.982,Z 169,A -110.1611,B 9.5896,C 0.3721,E1 9.5368,E2 201.4943} C_DIS
LIN {X -55.3677,Y -127.6581,Z 169,A -111.6742,B 9.5896,C 0.3727,E1 9.5329,E2 203.0207} C_DIS
LIN {X -58.7447,Y -126.1401,Z 169,A -113.1442,B 9.5897,C 0.3699,E1 9.5292,E2 204.4838} C_DIS
LIN {X -64.1557,Y -123.4751,Z 169,A -116.0805,B 9.5895,C 0.376,E1 9.5217,E2 207.4778} C_DIS
LIN {X -68.0514,Y -121.3743,Z 169,A -117.3461,B 9.59,C 0.3626,E1 9.5188,E2 208.6723} C_DIS
LIN {X -71.0491,Y -119.6443,Z 169,A -118.953,B 9.59,C 0.3642,E1 9.5149,E2 210.3024} C_DIS
LIN {X -74.6949,Y -117.4032,Z 169,A -120.7869,B 9.59,C 0.3631,E1 9.5105,E2 212.1452} C_DIS
LIN {X -77.6941,Y -115.4402,Z 169,A -122.2537,B 9.59,C 0.3607,E1 9.5071,E2 213.6106} C_DIS
LIN {X -82.9364,Y -111.7322,Z 169,A -125.013,B 9.5902,C 0.3587,E1 9.5008,E2 216.3841} C_DIS
LIN {X -87.0432,Y -108.5648,Z 169,A -127.0871,B 9.5903,C 0.3538,E1 9.4963,E2 218.45} C_DIS
LIN {X -90.5221,Y -105.6814,Z 169,A -129.0062,B 9.5904,C 0.3516,E1 9.4922,E2 220.3761} C_DIS
LIN {X -93.7409,Y -102.8369,Z 169,A -130.734,B 9.5906,C 0.3475,E1 9.4886,E2 222.0981} C_DIS
LIN {X -97.1041,Y -99.6678,Z 169,A -132.6596,B 9.5906,C 0.3443,E1 9.4847,E2 224.026} C_DIS
LIN {X -99.5088,Y -97.2663,Z 169,A -133.9349,B 9.5909,C 0.3391,E1 9.4823,E2 225.285} C_DIS
LIN {X -103.3682,Y -93.1545,Z 169,A -136.872,B 9.5906,C 0.3459,E1 9.4766,E2 228.2991} C_DIS
LIN {X -106.4678,Y -89.5953,Z 169,A -138.2123,B 9.5912,C 0.3305,E1 9.4743,E2 229.5622} C_DIS
LIN {X -108.7401,Y -86.8235,Z 169,A -139.8861,B 9.5912,C 0.3309,E1 9.4713,E2 231.2605} C_DIS
LIN {X -111.7854,Y -82.8662,Z 169,A -141.8782,B 9.5913,C 0.3251,E1 9.4679,E2 233.2435} C_DIS
LIN {X -114.1789,Y -79.5354,Z 169,A -143.6671,B 9.5914,C 0.3231,E1 9.465,E2 235.0443} C_DIS
LIN {X -116.8163,Y -75.6087,Z 169,A -145.6096,B 9.5916,C 0.3183,E1 9.4621,E2 236.9851} C_DIS
LIN {X -119.2449,Y -71.7179,Z 169,A -147.6574,B 9.5916,C 0.3167,E1 9.459,E2 239.0519} C_DIS
LIN {X -121.7692,Y -67.3422,Z 169,A -149.8998,B 9.5916,C 0.3145,E1 9.4559,E2 241.3135} C_DIS
LIN {X -123.392,Y -64.3173,Z 169,A -150.9931,B 9.592,C 0.305,E1 9.4546,E2 242.3654} C_DIS
LIN {X -124.9085,Y -61.3193,Z 169,A -152.4014,B 9.592,C 0.302,E1 9.4528,E2 243.776} C_DIS
LIN {X -126.4339,Y -58.1093,Z 169,A -153.8869,B 9.5922,C 0.2986,E1 9.4511,E2 245.2633} C_DIS
LIN {X -127.8157,Y -55.0032,Z 169,A -155.3198,B 9.5922,C 0.2955,E1 9.4495,E2 246.6994} C_DIS
LIN {X -129.377,Y -51.2292,Z 169,A -157.291,B 9.5922,C 0.2963,E1 9.4474,E2 248.706} C_DIS
LIN {X -130.9773,Y -46.9803,Z 169,A -158.9279,B 9.5926,C 0.287,E1 9.4458,E2 250.3121} C_DIS
LIN {X -132.1124,Y -43.6872,Z 169,A -160.3119,B 9.5926,C 0.2822,E1 9.4446,E2 251.6886} C_DIS
LIN {X -133.0699,Y -40.6766,Z 169,A -162.0429,B 9.5926,C 0.2863,E1 9.4431,E2 253.4727} C_DIS
LIN {X -134.1112,Y -37.1016,Z 169,A -163.2038,B 9.5929,C 0.2754,E1 9.4423,E2 254.5856} C_DIS
LIN {X -134.9035,Y -34.1065,Z 169,A -164.5365,B 9.5929,C 0.2729,E1 9.4413,E2 255.9245} C_DIS
LIN {X -135.6765,Y -30.8883,Z 169,A -165.969,B 9.593,C 0.2703,E1 9.4404,E2 257.3646} C_DIS
LIN {X -136.621,Y -26.4006,Z 169,A -167.867,B 9.5932,C 0.2651,E1 9.4394,E2 259.2623} C_DIS
LIN {X -137.2614,Y -22.8369,Z 169,A -169.3368,B 9.5933,C 0.2605,E1 9.4387,E2 260.7281} C_DIS
LIN {X -137.7845,Y -19.435,Z 169,A -170.7757,B 9.5933,C 0.2568,E1 9.4381,E2 262.1685} C_DIS
LIN {X -138.2613,Y -15.7058,Z 169,A -172.5108,B 9.5934,C 0.2557,E1 9.4375,E2 263.9257} C_DIS
LIN {X -138.6749,Y -11.4707,Z 169,A -174.0977,B 9.5936,C 0.2477,E1 9.4371,E2 265.4903} C_DIS
LIN {X -138.9221,Y -7.9545,Z 169,A -175.9074,B 9.5936,C 0.2498,E1 9.4368,E2 267.3435} C_DIS
LIN {X -139.0746,Y -4.588,Z 169,A -177.0873,B 9.5938,C 0.2421,E1 9.4367,E2 268.4962} C_DIS
LIN {X -139.1311,Y 2.2012,Z 169,A -179.8538,B 9.594,C 0.2335,E1 9.4367,E2 271.2563} C_DIS
LIN {X -139.0213,Y 5.9722,Z 169,A 178.2795,B 9.594,C 0.2345,E1 9.4368,E2 273.1607} C_DIS
LIN {X -138.8412,Y 9.268,Z 169,A 177.2113,B 9.5942,C 0.2254,E1 9.437,E2 274.1912} C_DIS
LIN {X -138.5132,Y 13.2797,Z 169,A 175.5248,B 9.5942,C 0.2211,E1 9.4374,E2 275.8797} C_DIS
LIN {X -138.1853,Y 16.3425,Z 169,A 174.1771,B 9.5943,C 0.2188,E1 9.4379,E2 277.236} C_DIS
LIN {X -137.7379,Y 19.7614,Z 169,A 172.7826,B 9.5944,C 0.2143,E1 9.4384,E2 278.626} C_DIS
LIN {X -137.2358,Y 22.9903,Z 169,A 171.4127,B 9.5945,C 0.2108,E1 9.439,E2 279.9975} C_DIS
LIN {X -136.6128,Y 26.4437,Z 169,A 169.9648,B 9.5945,C 0.2067,E1 9.4397,E2 281.4443} C_DIS
LIN {X -135.9707,Y 29.5669,Z 169,A 168.5848,B 9.5947,C 0.2041,E1 9.4405,E2 282.8313} C_DIS
LIN {X -135.0864,Y 33.384,Z 169,A 166.819,B 9.5947,C 0.2023,E1 9.4417,E2 284.6145} C_DIS
LIN {X -133.9914,Y 37.5299,Z 169,A 165.1225,B 9.5948,C 0.196,E1 9.4429,E2 286.3004} C_DIS
LIN {X -132.8382,Y 41.4335,Z 169,A 163.4802,B 9.5949,C 0.1908,E1 9.4443,E2 287.9368} C_DIS
LIN {X -131.7765,Y 44.6958,Z 169,A 162.0422,B 9.5949,C 0.1873,E1 9.4455,E2 289.3766} C_DIS
LIN {X -130.5533,Y 48.1507,Z 169,A 160.1574,B 9.5949,C 0.1898,E1 9.4474,E2 291.3064} C_DIS
LIN {X -129.2856,Y 51.4563,Z 169,A 159.0829,B 9.5951,C 0.179,E1 9.4484,E2 292.3318} C_DIS
LIN {X -127.8512,Y 54.9209,Z 169,A 157.3963,B 9.5951,C 0.1774,E1 9.4503,E2 294.0345} C_DIS
LIN {X -126.1524,Y 58.7182,Z 169,A 155.6979,B 9.5953,C 0.1725,E1 9.4522,E2 295.7292} C_DIS
LIN {X -124.389,Y 62.3715,Z 169,A 153.8775,B 9.5953,C 0.1708,E1 9.4545,E2 297.5665} C_DIS
LIN {X -122.3468,Y 66.288,Z 169,A 152.0686,B 9.5953,C 0.1659,E1 9.4569,E2 299.3722} C_DIS
LIN {X -119.3499,Y 71.5431,Z 169,A 149.4079,B 9.5954,C 0.1627,E1 9.4606,E2 302.0514} C_DIS
LIN {X -116.7133,Y 75.7674,Z 169,A 147.7159,B 9.5956,C 0.1511,E1 9.4631,E2 303.6967} C_DIS
LIN {X -114.9313,Y 78.4449,Z 169,A 146.1166,B 9.5956,C 0.1528,E1 9.4656,E2 305.3288} C_DIS
LIN {X -112.3702,Y 82.0717,Z 169,A 144.2452,B 9.5956,C 0.1492,E1 9.4687,E2 307.2036} C_DIS
LIN {X -108.7847,Y 86.7675,Z 169,A 142.0798,B 9.5958,C 0.1387,E1 9.4723,E2 309.3333} C_DIS
LIN {X -106.8461,Y 89.1445,Z 169,A 140.5258,B 9.5958,C 0.1411,E1 9.4751,E2 310.9221} C_DIS
LIN {X -103.3981,Y 93.1212,Z 169,A 138.0925,B 9.5958,C 0.1412,E1 9.4797,E2 313.3861} C_DIS
LIN {X -100.9034,Y 95.8195,Z 169,A 136.8972,B 9.5959,C 0.1321,E1 9.4819,E2 314.5406} C_DIS
LIN {X -97.9928,Y 98.7933,Z 169,A 134.5718,B 9.5958,C 0.1398,E1 9.4867,E2 316.9396} C_DIS
LIN {X -94.3573,Y 102.2715,Z 169,A 132.9882,B 9.596,C 0.1266,E1 9.4898,E2 318.4612} C_DIS
LIN {X -91.1327,Y 105.1556,Z 169,A 131.1548,B 9.596,C 0.1241,E1 9.4936,E2 320.2993} C_DIS
LIN {X -87.5637,Y 108.1451,Z 169,A 128.981,B 9.596,C 0.1253,E1 9.4984,E2 322.5029} C_DIS
LIN {X -84.6465,Y 110.4431,Z 169,A 127.5032,B 9.596,C 0.1216,E1 9.5016,E2 323.9729} C_DIS
LIN {X -81.9265,Y 112.4759,Z 169,A 126.5937,B 9.5962,C 0.11,E1 9.5035,E2 324.8208} C_DIS
LIN {X -78.658,Y 114.785,Z 169,A 124.882,B 9.5962,C 0.1084,E1 9.5075,E2 326.5389} C_DIS
LIN {X -76.0326,Y 116.5411,Z 169,A 123.0419,B 9.5962,C 0.1165,E1 9.5119,E2 328.4444} C_DIS
LIN {X -72.8607,Y 118.5497,Z 169,A 120.9997,B 9.596,C 0.1234,E1 9.5169,E2 330.5459} C_DIS
LIN {X -67.343,Y 121.7687,Z 169,A 119.2742,B 9.5963,C 0.1024,E1 9.5209,E2 332.1582} C_DIS
LIN {X -64.3034,Y 123.3993,Z 169,A 117.7846,B 9.5963,C 0.1017,E1 9.5245,E2 333.6551} C_DIS
LIN {X -60.9755,Y 125.0781,Z 169,A 116.1352,B 9.5963,C 0.1019,E1 9.5287,E2 335.3174} C_DIS
LIN {X -57.4107,Y 126.754,Z 169,A 114.6783,B 9.5963,C 0.0967,E1 9.5323,E2 336.7526} C_DIS
LIN {X -54.8176,Y 127.8959,Z 169,A 113.4361,B 9.5963,C 0.0967,E1 9.5355,E2 338.0031} C_DIS
LIN {X -50.011,Y 129.8508,Z 169,A 111.6259,B 9.5964,C 0.088,E1 9.5401,E2 339.7712} C_DIS
LIN {X -44.5253,Y 131.8333,Z 169,A 108.9617,B 9.5964,C 0.0908,E1 9.5472,E2 342.4664} C_DIS
LIN {X -40.7239,Y 133.0554,Z 169,A 107.1832,B 9.5964,C 0.0919,E1 9.552,E2 344.2604} C_DIS
LIN {X -37.2522,Y 134.069,Z 169,A 105.7287,B 9.5964,C 0.09,E1 9.5559,E2 345.7095} C_DIS
LIN {X -33.9129,Y 134.9526,Z 169,A 104.2752,B 9.5964,C 0.0895,E1 9.5598,E2 347.1659} C_DIS
LIN {X -29.9716,Y 135.8834,Z 169,A 102.4353,B 9.5964,C 0.0918,E1 9.5649,E2 349.026} C_DIS
LIN {X -25.4789,Y 136.7972,Z 169,A 100.8121,B 9.5964,C 0.0854,E1 9.5692,E2 350.6153} C_DIS
LIN {X -20.4474,Y 137.6381,Z 169,A 98.4682,B 9.5964,C 0.0893,E1 9.5758,E2 352.988} C_DIS
LIN {X -16.2103,Y 138.2011,Z 169,A 96.3397,B 9.5964,C 0.0961,E1 9.5818,E2 355.1609} C_DIS
LIN {X -11.7453,Y 138.6518,Z 169,A 94.8651,B 9.5964,C 0.088,E1 9.5858,E2 356.5886} C_DIS
LIN {X -5.1543,Y 139.0532,Z 169,A 92.3391,B 9.5964,C 0.0835,E1 9.5927,E2 359.0894} C_DIS
LIN {X -2.1484,Y 139.132,Z 169,A 90.9575,B 9.5964,C 0.0864,E1 9.5966,E2 360.4882} C_DIS
LIN {X 2.063,Y 139.1334,Z 169,A 89.0002,B 9.5964,C 0.091,E1 9.6022,E2 362.4722} C_DIS
LIN {X 5.42,Y 139.0428,Z 169,A 87.6055,B 9.5964,C 0.0913,E1 9.6061,E2 363.8678} C_DIS
LIN {X 8.894,Y 138.8643,Z 169,A 86.4834,B 9.5964,C 0.0851,E1 9.6091,E2 364.951} C_DIS
LIN {X 13.0603,Y 138.5343,Z 169,A 84.3644,B 9.5964,C 0.0938,E1 9.6151,E2 367.1185} C_DIS
LIN {X 17.0478,Y 138.1012,Z 169,A 83.1415,B 9.5964,C 0.0853,E1 9.6184,E2 368.288} C_DIS
LIN {X 21.9542,Y 137.407,Z 169,A 81.0997,B 9.5964,C 0.0862,E1 9.624,E2 370.3294} C_DIS
LIN {X 24.8672,Y 136.9086,Z 169,A 79.6173,B 9.5964,C 0.0924,E1 9.6282,E2 371.8443} C_DIS
LIN {X 32.8145,Y 135.2237,Z 169,A 76.5375,B 9.5964,C 0.0887,E1 9.6365,E2 374.8903} C_DIS
LIN {X 35.7272,Y 134.4834,Z 169,A 75.2388,B 9.5964,C 0.0909,E1 9.64,E2 376.1964} C_DIS
LIN {X 39.453,Y 133.4383,Z 169,A 73.7244,B 9.5964,C 0.0904,E1 9.6441,E2 377.7008} C_DIS
LIN {X 43.1095,Y 132.3041,Z 169,A 72.0041,B 9.5964,C 0.0949,E1 9.6487,E2 379.4388} C_DIS
LIN {X 46.9968,Y 130.9714,Z 169,A 70.4183,B 9.5964,C 0.0942,E1 9.6528,E2 381.0111} C_DIS
LIN {X 50.3093,Y 129.7349,Z 169,A 69.0229,B 9.5964,C 0.0942,E1 9.6564,E2 382.3988} C_DIS
LIN {X 54.361,Y 128.092,Z 169,A 67.2491,B 9.5964,C 0.0957,E1 9.661,E2 384.1693} C_DIS
LIN {X 57.0578,Y 126.9118,Z 169,A 65.7653,B 9.5963,C 0.103,E1 9.6649,E2 385.6867} C_DIS
LIN {X 65.2155,Y 122.9203,Z 169,A 62.5015,B 9.5963,C 0.0972,E1 9.6729,E2 388.8914} C_DIS
LIN {X 67.9997,Y 121.4033,Z 169,A 60.9037,B 9.5963,C 0.1056,E1 9.6769,E2 390.5259} C_DIS
LIN {X 72.044,Y 119.0477,Z 169,A 58.988,B 9.5963,C 0.1081,E1 9.6815,E2 392.4403} C_DIS
LIN {X 76.0167,Y 116.5514,Z 169,A 56.7591,B 9.5961,C 0.1178,E1 9.6868,E2 394.7064} C_DIS
LIN {X 79.3216,Y 114.3266,Z 169,A 55.0692,B 9.5961,C 0.1215,E1 9.6907,E2 396.4026} C_DIS
LIN {X 82.9391,Y 111.7311,Z 169,A 53.6377,B 9.5961,C 0.1156,E1 9.6938,E2 397.7846} C_DIS
LIN {X 86.5591,Y 108.9505,Z 169,A 51.9466,B 9.5961,C 0.1146,E1 9.6975,E2 399.4526} C_DIS
LIN {X 90.3712,Y 105.8103,Z 169,A 50.0039,B 9.5961,C 0.1162,E1 9.7016,E2 401.3845} C_DIS
LIN {X 92.7662,Y 103.7165,Z 169,A 48.4663,B 9.5961,C 0.1239,E1 9.7049,E2 402.951} C_DIS
LIN {X 96.9444,Y 99.8224,Z 169,A 46.147,B 9.596,C 0.1278,E1 9.7096,E2 405.2669} C_DIS
LIN {X 100.15,Y 96.606,Z 169,A 43.6008,B 9.5957,C 0.1472,E1 9.7147,E2 407.898} C_DIS
LIN {X 104.263,Y 92.1516,Z 169,A 42.2364,B 9.596,C 0.1264,E1 9.717,E2 409.1221} C_DIS
LIN {X 107.5731,Y 88.2654,Z 169,A 39.8321,B 9.5958,C 0.138,E1 9.7214,E2 411.5653} C_DIS
LIN {X 111.0989,Y 83.7837,Z 169,A 37.501,B 9.5958,C 0.143,E1 9.7254,E2 413.8955} C_DIS
LIN {X 113.4896,Y 80.5167,Z 169,A 35.7645,B 9.5957,C 0.1485,E1 9.7283,E2 415.6416} C_DIS
LIN {X 116.0957,Y 76.7107,Z 169,A 33.9012,B 9.5957,C 0.1522,E1 9.7312,E2 417.5014} C_DIS
LIN {X 119.1077,Y 71.9447,Z 169,A 31.5817,B 9.5955,C 0.1578,E1 9.7346,E2 419.822} C_DIS
LIN {X 121.3877,Y 68.0276,Z 169,A 29.8032,B 9.5955,C 0.1604,E1 9.737,E2 421.5905} C_DIS
LIN {X 123.3919,Y 64.3174,Z 169,A 28.1543,B 9.5955,C 0.1628,E1 9.7392,E2 423.2294} C_DIS
LIN {X 124.9415,Y 61.2525,Z 169,A 26.706,B 9.5954,C 0.1672,E1 9.741,E2 424.683} C_DIS
LIN {X 126.4503,Y 58.074,Z 169,A 25.2882,B 9.5954,C 0.1703,E1 9.7427,E2 426.0979} C_DIS
LIN {X 128.8431,Y 52.5541,Z 169,A 22.2489,B 9.5949,C 0.1903,E1 9.746,E2 429.2095} C_DIS
LIN {X 130.7316,Y 47.6617,Z 169,A 20.8885,B 9.5952,C 0.177,E1 9.7473,E2 430.471} C_DIS
LIN {X 132.0926,Y 43.7465,Z 169,A 19.0846,B 9.5951,C 0.184,E1 9.7489,E2 432.2885} C_DIS
LIN {X 133.1322,Y 40.473,Z 169,A 17.6766,B 9.595,C 0.1878,E1 9.7501,E2 433.6968} C_DIS
LIN {X 134.0903,Y 37.1764,Z 169,A 16.2506,B 9.5949,C 0.192,E1 9.7512,E2 435.1255} C_DIS
LIN {X 135.2084,Y 32.8782,Z 169,A 14.4261,B 9.5948,C 0.1971,E1 9.7524,E2 436.9509} C_DIS
LIN {X 136.256,Y 28.227,Z 169,A 12.3709,B 9.5946,C 0.2049,E1 9.7536,E2 439.0195} C_DIS
LIN {X 137.2591,Y 22.8507,Z 169,A 9.9614,B 9.5944,C 0.2151,E1 9.7548,E2 441.4507} C_DIS
LIN {X 137.8512,Y 18.9688,Z 169,A 8.7725,B 9.5945,C 0.2094,E1 9.7553,E2 442.587} C_DIS
LIN {X 138.5263,Y 13.1428,Z 169,A 6.3571,B 9.5944,C 0.2164,E1 9.756,E2 445.0046} C_DIS
LIN {X 138.8363,Y 9.3442,Z 169,A 4.6674,B 9.5942,C 0.2239,E1 9.7563,E2 446.7112} C_DIS
LIN {X 139.1133,Y 3.188,Z 169,A 2.0554,B 9.594,C 0.2331,E1 9.7566,E2 449.335} C_DIS
LIN {X 139.1517,Y -0.1637,Z 169,A 0.8721,B 9.594,C 0.2323,E1 9.7566,E2 450.4947} C_DIS
LIN {X 139.1002,Y -3.6688,Z 169,A -0.4802,B 9.594,C 0.2343,E1 9.7566,E2 451.8367} C_DIS
LIN {X 138.9359,Y -7.7228,Z 169,A -2.3414,B 9.5937,C 0.2438,E1 9.7563,E2 453.7239} C_DIS
LIN {X 138.3109,Y -15.2472,Z 169,A -5.1994,B 9.5937,C 0.2468,E1 9.7556,E2 456.553} C_DIS
LIN {X 137.4165,Y -21.8925,Z 169,A -7.8327,B 9.5935,C 0.2517,E1 9.7545,E2 459.1728} C_DIS
LIN {X 136.0054,Y -29.4064,Z 169,A -10.9882,B 9.5933,C 0.2609,E1 9.7529,E2 462.3326} C_DIS
LIN {X 135.2428,Y -32.7355,Z 169,A -12.5695,B 9.5931,C 0.2692,E1 9.7518,E2 463.9377} C_DIS
LIN {X 133.9667,Y -37.6183,Z 169,A -14.4831,B 9.5931,C 0.2711,E1 9.7504,E2 465.8325} C_DIS
LIN {X 132.885,Y -41.2806,Z 169,A -15.9396,B 9.593,C 0.2727,E1 9.7493,E2 467.276} C_DIS
LIN {X 131.9248,Y -44.2504,Z 169,A -17.249,B 9.5928,C 0.2769,E1 9.7481,E2 468.5898} C_DIS
LIN {X 130.7179,Y -47.6999,Z 169,A -19.2355,B 9.5924,C 0.2927,E1 9.7462,E2 470.6393} C_DIS
LIN {X 129.0978,Y -51.9222,Z 169,A -20.2853,B 9.5928,C 0.2782,E1 9.7452,E2 471.5872} C_DIS
LIN {X 128.0704,Y -54.4137,Z 169,A -22.5716,B 9.5919,C 0.3096,E1 9.7426,E2 474.025} C_DIS
LIN {X 125.2544,Y -60.6131,Z 169,A -24.4052,B 9.5923,C 0.2938,E1 9.7405,E2 475.7381} C_DIS
LIN {X 123.7792,Y -63.5695,Z 169,A -25.7799,B 9.5923,C 0.2977,E1 9.7387,E2 477.1161} C_DIS
LIN {X 121.8382,Y -67.2175,Z 169,A -27.5482,B 9.592,C 0.3038,E1 9.7364,E2 478.8949} C_DIS
LIN {X 119.9728,Y -70.4927,Z 169,A -29.0471,B 9.592,C 0.3065,E1 9.7343,E2 480.3886} C_DIS
LIN {X 117.5994,Y -74.3848,Z 169,A -30.9763,B 9.5918,C 0.3125,E1 9.7314,E2 482.3265} C_DIS
LIN {X 115.5011,Y -77.6038,Z 169,A -32.4493,B 9.5918,C 0.3138,E1 9.7292,E2 483.7872} C_DIS
LIN {X 112.001,Y -82.5743,Z 169,A -34.7845,B 9.5917,C 0.3159,E1 9.7254,E2 486.1035} C_DIS
LIN {X 108.2155,Y -87.4763,Z 169,A -37.2872,B 9.5915,C 0.3208,E1 9.7212,E2 488.6028} C_DIS
LIN {X 105.8561,Y -90.3174,Z 169,A -39.0836,B 9.5912,C 0.3309,E1 9.7178,E2 490.4363} C_DIS
LIN {X 102.0586,Y -94.5877,Z 169,A -41.6088,B 9.5908,C 0.3402,E1 9.713,E2 492.986} C_DIS
LIN {X 99.3097,Y -97.4693,Z 169,A -42.8872,B 9.591,C 0.3352,E1 9.7106,E2 494.2197} C_DIS
LIN {X 96.1912,Y -100.5482,Z 169,A -44.6858,B 9.5909,C 0.3389,E1 9.707,E2 496.0193} C_DIS
LIN {X 92.0616,Y -104.3426,Z 169,A -47.3297,B 9.5904,C 0.3514,E1 9.7014,E2 498.7085} C_DIS
LIN {X 88.885,Y -107.0615,Z 169,A -48.4002,B 9.5909,C 0.3395,E1 9.6993,E2 499.6969} C_DIS
LIN {X 86.5949,Y -108.9221,Z 169,A -49.8742,B 9.5906,C 0.348,E1 9.6961,E2 501.2056} C_DIS
LIN {X 82.8177,Y -111.8215,Z 169,A -51.5834,B 9.5906,C 0.3457,E1 9.6923,E2 502.8843} C_DIS
LIN {X 78.0524,Y -115.1977,Z 169,A -53.9001,B 9.5906,C 0.3479,E1 9.6871,E2 505.1919} C_DIS
LIN {X 75.682,Y -116.7687,Z 169,A -55.736,B 9.5899,C 0.3653,E1 9.6826,E2 507.1145} C_DIS
LIN {X 72.0748,Y -119.0291,Z 169,A -57.2951,B 9.5899,C 0.3637,E1 9.6789,E2 508.6504} C_DIS
LIN {X 69.2323,Y -120.705,Z 169,A -58.2885,B 9.5902,C 0.3574,E1 9.6766,E2 509.598} C_DIS
LIN {X 65.5458,Y -122.746,Z 169,A -60.0906,B 9.5901,C 0.3616,E1 9.6722,E2 511.4103} C_DIS
LIN {X 62.8563,Y -124.1423,Z 169,A -61.3458,B 9.59,C 0.3635,E1 9.669,E2 512.6674} C_DIS
LIN {X 59.1389,Y -125.9578,Z 169,A -63.2614,B 9.5897,C 0.3707,E1 9.6641,E2 514.6119} C_DIS
LIN {X 53.3663,Y -128.5078,Z 169,A -65.6282,B 9.5897,C 0.3687,E1 9.6581,E2 516.9509} C_DIS
LIN {X 50.0529,Y -129.8346,Z 169,A -67.0522,B 9.5897,C 0.3694,E1 9.6544,E2 518.3702} C_DIS
LIN {X 46.4749,Y -131.1596,Z 169,A -69.1269,B 9.5892,C 0.3825,E1 9.6488,E2 520.511} C_DIS
LIN {X 42.3031,Y -132.5617,Z 169,A -70.0922,B 9.5899,C 0.3653,E1 9.6466,E2 521.3684} C_DIS
LIN {X 38.8204,Y -133.6235,Z 169,A -71.9387,B 9.5896,C 0.3745,E1 9.6415,E2 523.261} C_DIS
LIN {X 35.463,Y -134.5538,Z 169,A -73.7044,B 9.5892,C 0.3832,E1 9.6366,E2 525.0704} C_DIS
LIN {X 31.7313,Y -135.484,Z 169,A -75.0389,B 9.5894,C 0.3789,E1 9.6331,E2 526.374} C_DIS
LIN {X 27.577,Y -136.3882,Z 169,A -77.3106,B 9.5889,C 0.3916,E1 9.6267,E2 528.7136} C_DIS
LIN {X 22.2974,Y -137.3515,Z 169,A -78.8352,B 9.5894,C 0.378,E1 9.6227,E2 530.1518} C_DIS
LIN {X 16.0649,Y -138.2184,Z 169,A -81.3667,B 9.5894,C 0.378,E1 9.6157,E2 532.6771} C_DIS
LIN {X 13.1476,Y -138.5259,Z 169,A -82.6856,B 9.5894,C 0.3809,E1 9.612,E2 534.0111} C_DIS
LIN {X 9.1642,Y -138.8476,Z 169,A -84.4689,B 9.5892,C 0.3845,E1 9.607,E2 535.813} C_DIS
LIN {X 2.5363,Y -139.1255,Z 169,A -87.0512,B 9.5892,C 0.3818,E1 9.5998,E2 538.3775} C_DIS
LIN {X 2.5363,Y -139.1255,Z 169,A -87.0512,B 9.5892,C 0.3818,E1 9.5998,E2 538.3775} C_DIS
Enddeposition()
LIN {X 1.016,Y -140.0559,Z 169,A -87.5607,B 9.5893,C 0.3851,E1 9.5985,E2 538.9066} C_DIS
Startdeposition()
$VEL.CP = VEL_PRINT
LIN {X 5.0028,Y -139.9721,Z 169,A -85.337,B 9.5899,C 0.3719,E1 9.605,E2 536.6047} C_DIS
LIN {X 8.9547,Y -139.7746,Z 169,A -83.7515,B 9.5899,C 0.3721,E1 9.6094,E2 535.0227} C_DIS
LIN {X 12.8608,Y -139.47,Z 169,A -82.2708,B 9.5898,C 0.3743,E1 9.6135,E2 533.5572} C_DIS
LIN {X 16.2263,Y -139.118,Z 169,A -80.6133,B 9.59,C 0.3675,E1 9.6182,E2 531.8629} C_DIS
LIN {X 20.5345,Y -138.5491,Z 169,A -78.9731,B 9.59,C 0.3697,E1 9.6226,E2 530.2398} C_DIS
LIN {X 26.8729,Y -137.4596,Z 169,A -76.2553,B 9.59,C 0.3661,E1 9.6302,E2 527.5089} C_DIS
LIN {X 30.9491,Y -136.5985,Z 169,A -74.8479,B 9.5899,C 0.3715,E1 9.6339,E2 526.1393} C_DIS
LIN {X 35.9338,Y -135.3725,Z 169,A -72.5838,B 9.5901,C 0.3661,E1 9.6401,E2 523.8523} C_DIS
LIN {X 39.2694,Y -134.4427,Z 169,A -71.2012,B 9.5901,C 0.3655,E1 9.6438,E2 522.4731} C_DIS
LIN {X 42.4395,Y -133.4759,Z 169,A -69.5465,B 9.5904,C 0.3573,E1 9.6483,E2 520.778} C_DIS
LIN {X 45.5738,Y -132.4388,Z 169,A -68.4602,B 9.5902,C 0.362,E1 9.6511,E2 519.7256} C_DIS
LIN {X 48.9843,Y -131.2153,Z 169,A -67.0058,B 9.5902,C 0.361,E1 9.6549,E2 518.2737} C_DIS
LIN {X 52.4567,Y -129.866,Z 169,A -65.5394,B 9.5902,C 0.3605,E1 9.6587,E2 516.8136} C_DIS
LIN {X 59.0449,Y -127.0065,Z 169,A -62.583,B 9.5904,C 0.3563,E1 9.6663,E2 513.8525} C_DIS
LIN {X 62.5557,Y -125.3159,Z 169,A -60.8878,B 9.5906,C 0.3517,E1 9.6705,E2 512.1427} C_DIS
LIN {X 66.0004,Y -123.5374,Z 169,A -59.2918,B 9.5907,C 0.3492,E1 9.6745,E2 510.544} C_DIS
LIN {X 68.9839,Y -121.8967,Z 169,A -57.5435,B 9.5911,C 0.3386,E1 9.6789,E2 508.7475} C_DIS
LIN {X 72.8574,Y -119.622,Z 169,A -55.5133,B 9.5913,C 0.3311,E1 9.6837,E2 506.69} C_DIS
LIN {X 77.6042,Y -116.5978,Z 169,A -54.13,B 9.5907,C 0.349,E1 9.6867,E2 505.4261} C_DIS
LIN {X 80.7008,Y -114.4762,Z 169,A -52.333,B 9.591,C 0.3401,E1 9.6909,E2 503.5933} C_DIS
LIN {X 84.1626,Y -111.956,Z 169,A -50.5887,B 9.5911,C 0.3371,E1 9.6948,E2 501.8483} C_DIS
LIN {X 87.6537,Y -109.2446,Z 169,A -48.7755,B 9.5913,C 0.3335,E1 9.6988,E2 500.0327} C_DIS
LIN {X 90.1562,Y -107.1882,Z 169,A -47.5187,B 9.5913,C 0.3326,E1 9.7015,E2 498.7836} C_DIS
LIN {X 93.4579,Y -104.3218,Z 169,A -45.7598,B 9.5913,C 0.3297,E1 9.7052,E2 497.0268} C_DIS
LIN {X 96.3693,Y -101.6391,Z 169,A -44.1215,B 9.5915,C 0.3259,E1 9.7085,E2 495.3845} C_DIS
LIN {X 99.5269,Y -98.5489,Z 169,A -42.5076,B 9.5915,C 0.3267,E1 9.7117,E2 493.7941} C_DIS
LIN {X 101.7816,Y -96.2182,Z 169,A -40.9153,B 9.5918,C 0.3174,E1 9.7148,E2 492.1655} C_DIS
LIN {X 105.2413,Y -92.4223,Z 169,A -38.9075,B 9.5918,C 0.3149,E1 9.7185,E2 490.1678} C_DIS
LIN {X 108.0535,Y -89.1176,Z 169,A -37.2395,B 9.5919,C 0.3134,E1 9.7215,E2 488.512} C_DIS
LIN {X 111.4995,Y -84.7661,Z 169,A -34.8675,B 9.5922,C 0.3056,E1 9.7256,E2 486.1243} C_DIS
LIN {X 115.1113,Y -79.7926,Z 169,A -32.4092,B 9.5923,C 0.3008,E1 9.7296,E2 483.6708} C_DIS
LIN {X 117.4175,Y -76.3581,Z 169,A -30.7713,B 9.5924,C 0.298,E1 9.7321,E2 482.0382} C_DIS
LIN {X 119.8796,Y -72.4314,Z 169,A -28.9707,B 9.5924,C 0.2955,E1 9.7347,E2 480.2481} C_DIS
LIN {X 121.8714,Y -69.0288,Z 169,A -27.2927,B 9.5927,C 0.2897,E1 9.737,E2 478.5599} C_DIS
LIN {X 123.8955,Y -65.321,Z 169,A -25.7507,B 9.5927,C 0.2897,E1 9.739,E2 477.0403} C_DIS
LIN {X 125.4424,Y -62.2994,Z 169,A -24.3416,B 9.5927,C 0.2856,E1 9.7408,E2 475.627} C_DIS
LIN {X 127.8001,Y -57.3064,Z 169,A -22.1359,B 9.5929,C 0.2809,E1 9.7434,E2 473.4259} C_DIS
LIN {X 129.1673,Y -54.1548,Z 169,A -20.7427,B 9.593,C 0.2773,E1 9.7449,E2 472.0328} C_DIS
LIN {X 130.4409,Y -51.0113,Z 169,A -19.5692,B 9.593,C 0.2788,E1 9.7461,E2 470.8857} C_DIS
LIN {X 131.7252,Y -47.596,Z 169,A -18.0871,B 9.593,C 0.2749,E1 9.7476,E2 469.4034} C_DIS
LIN {X 132.7848,Y -44.5556,Z 169,A -16.5656,B 9.5933,C 0.2662,E1 9.749,E2 467.8539} C_DIS
LIN {X 133.7396,Y -41.6057,Z 169,A -14.8564,B 9.5937,C 0.2517,E1 9.7505,E2 466.0855} C_DIS
LIN {X 134.9812,Y -37.3781,Z 169,A -13.5838,B 9.5935,C 0.2598,E1 9.7514,E2 464.8805} C_DIS
LIN {X 136.3241,Y -32.1427,Z 169,A -11.2655,B 9.5938,C 0.2508,E1 9.7529,E2 462.546} C_DIS
LIN {X 137.2658,Y -27.8401,Z 169,A -9.5546,B 9.5938,C 0.2479,E1 9.7539,E2 460.8449} C_DIS
LIN {X 138.0814,Y -23.4664,Z 169,A -7.9806,B 9.5938,C 0.2488,E1 9.7547,E2 459.3012} C_DIS
LIN {X 138.6177,Y -20.0539,Z 169,A -6.4081,B 9.594,C 0.2407,E1 9.7553,E2 457.7064} C_DIS
LIN {X 139.1103,Y -16.2907,Z 169,A -4.8267,B 9.5941,C 0.2355,E1 9.7559,E2 456.1198} C_DIS
LIN {X 139.5708,Y -11.7042,Z 169,A -3.0241,B 9.5942,C 0.2321,E1 9.7563,E2 454.3261} C_DIS
LIN {X 139.856,Y -7.5906,Z 169,A -1.3394,B 9.5943,C 0.2272,E1 9.7566,E2 452.64} C_DIS
LIN {X 140.0059,Y -3.9195,Z 169,A 0.0707,B 9.5943,C 0.2251,E1 9.7568,E2 451.2406} C_DIS
LIN {X 140.0647,Y -0.0833,Z 169,A 1.862,B 9.5946,C 0.2151,E1 9.7568,E2 449.4189} C_DIS
LIN {X 139.9849,Y 4.6704,Z 169,A 3.6763,B 9.5946,C 0.2126,E1 9.7567,E2 447.6197} C_DIS
LIN {X 139.7771,Y 8.9136,Z 169,A 5.3461,B 9.5947,C 0.2093,E1 9.7564,E2 445.9571} C_DIS
LIN {X 139.36,Y 14.006,Z 169,A 7.524,B 9.5949,C 0.201,E1 9.7558,E2 443.7659} C_DIS
LIN {X 138.7249,Y 19.3043,Z 169,A 10.0194,B 9.5952,C 0.187,E1 9.7549,E2 441.2279} C_DIS
LIN {X 137.983,Y 24.0429,Z 169,A 11.5096,B 9.5951,C 0.1931,E1 9.7542,E2 439.7974} C_DIS
LIN {X 137.2779,Y 27.7803,Z 169,A 13.3915,B 9.5953,C 0.1806,E1 9.7532,E2 437.8718} C_DIS
LIN {X 136.3449,Y 32.0566,Z 169,A 14.7801,B 9.5953,C 0.1855,E1 9.7523,E2 436.5339} C_DIS
LIN {X 135.5182,Y 35.3875,Z 169,A 16.2014,B 9.5953,C 0.1811,E1 9.7513,E2 435.1093} C_DIS
LIN {X 134.4762,Y 39.1551,Z 169,A 17.6859,B 9.5953,C 0.1794,E1 9.7502,E2 433.6383} C_DIS
LIN {X 133.3475,Y 42.8416,Z 169,A 19.2598,B 9.5954,C 0.1752,E1 9.7489,E2 432.0636} C_DIS
LIN {X 131.9459,Y 46.9839,Z 169,A 20.9057,B 9.5954,C 0.1738,E1 9.7474,E2 430.4348} C_DIS
LIN {X 130.5125,Y 50.8271,Z 169,A 23.2991,B 9.5958,C 0.1517,E1 9.7449,E2 427.9474} C_DIS
LIN {X 128.4385,Y 55.8616,Z 169,A 24.8791,B 9.5956,C 0.1617,E1 9.7433,E2 426.4499} C_DIS
LIN {X 126.1597,Y 60.8346,Z 169,A 27.1876,B 9.5958,C 0.1541,E1 9.7405,E2 424.1308} C_DIS
LIN {X 124.1408,Y 64.8538,Z 169,A 28.8545,B 9.5958,C 0.1536,E1 9.7384,E2 422.4849} C_DIS
LIN {X 122.0603,Y 68.693,Z 169,A 30.5885,B 9.5958,C 0.1503,E1 9.7361,E2 420.7567} C_DIS
LIN {X 117.6222,Y 76.0428,Z 169,A 34.3121,B 9.596,C 0.1367,E1 9.7306,E2 417.004} C_DIS
LIN {X 114.6962,Y 80.3889,Z 169,A 36.316,B 9.596,C 0.1349,E1 9.7275,E2 415.0169} C_DIS
LIN {X 112.0274,Y 84.0679,Z 169,A 38.2107,B 9.5961,C 0.1298,E1 9.7243,E2 413.1168} C_DIS
LIN {X 108.9481,Y 88.0213,Z 169,A 40.1399,B 9.5961,C 0.128,E1 9.721,E2 411.2022} C_DIS
LIN {X 106.0564,Y 91.4849,Z 169,A 41.8552,B 9.5961,C 0.1271,E1 9.7179,E2 409.5028} C_DIS
LIN {X 102.9706,Y 94.9449,Z 169,A 43.8443,B 9.5962,C 0.1209,E1 9.7142,E2 407.501} C_DIS
LIN {X 99.9597,Y 98.1096,Z 169,A 45.6158,B 9.5962,C 0.1175,E1 9.7107,E2 405.7308} C_DIS
LIN {X 96.7382,Y 101.2874,Z 169,A 47.4763,B 9.5963,C 0.1136,E1 9.707,E2 403.8685} C_DIS
LIN {X 93.2281,Y 104.5277,Z 169,A 49.386,B 9.5963,C 0.1109,E1 9.7031,E2 401.9639} C_DIS
LIN {X 89.6721,Y 107.5943,Z 169,A 51.3137,B 9.5964,C 0.1072,E1 9.6989,E2 400.0348} C_DIS
LIN {X 86.104,Y 110.4703,Z 169,A 53.1617,B 9.5964,C 0.1045,E1 9.6949,E2 398.1899} C_DIS
LIN {X 83.5175,Y 112.4379,Z 169,A 55.5732,B 9.5967,C 0.077,E1 9.6892,E2 395.6386} C_DIS
LIN {X 76.622,Y 117.2462,Z 169,A 57.8085,B 9.5965,C 0.0995,E1 9.6843,E2 393.5581} C_DIS
LIN {X 72.8713,Y 119.6135,Z 169,A 59.6769,B 9.5965,C 0.0955,E1 9.6799,E2 391.6826} C_DIS
LIN {X 69.0112,Y 121.8814,Z 169,A 61.5336,B 9.5965,C 0.0924,E1 9.6754,E2 389.8225} C_DIS
LIN {X 66.0676,Y 123.5013,Z 169,A 63.5144,B 9.5967,C 0.0767,E1 9.6703,E2 387.764} C_DIS
LIN {X 60.8883,Y 126.1341,Z 169,A 65.1906,B 9.5966,C 0.0896,E1 9.6663,E2 386.1775} C_DIS
LIN {X 57.4982,Y 127.7143,Z 169,A 66.5356,B 9.5966,C 0.092,E1 9.663,E2 384.8561} C_DIS
LIN {X 53.2182,Y 129.5584,Z 169,A 68.6668,B 9.5966,C 0.0849,E1 9.6574,E2 382.6965} C_DIS
LIN {X 49.5572,Y 131.0007,Z 169,A 70.0726,B 9.5966,C 0.0878,E1 9.6538,E2 381.3166} C_DIS
LIN {X 46.1757,Y 132.2301,Z 169,A 71.5098,B 9.5966,C 0.0871,E1 9.6501,E2 379.884} C_DIS
LIN {X 43.1643,Y 133.2444,Z 169,A 72.9902,B 9.5966,C 0.082,E1 9.6461,E2 378.3809} C_DIS
LIN {X 39.5736,Y 134.3536,Z 169,A 74.3302,B 9.5966,C 0.0851,E1 9.6425,E2 377.0661} C_DIS
LIN {X 36.337,Y 135.265,Z 169,A 75.6192,B 9.5966,C 0.086,E1 9.6391,E2 375.7883} C_DIS
LIN {X 30.2902,Y 136.748,Z 169,A 78.4316,B 9.5966,C 0.0786,E1 9.6314,E2 372.943} C_DIS
LIN {X 26.7037,Y 137.4919,Z 169,A 79.9014,B 9.5966,C 0.0784,E1 9.6274,E2 371.4773} C_DIS
LIN {X 23.7851,Y 138.0282,Z 169,A 81.333,B 9.5967,C 0.0731,E1 9.6234,E2 370.0184} C_DIS
LIN {X 20.5434,Y 138.5477,Z 169,A 82.5355,B 9.5967,C 0.0756,E1 9.6201,E2 368.8343} C_DIS
LIN {X 17.1523,Y 139.0076,Z 169,A 83.9206,B 9.5967,C 0.0754,E1 9.6163,E2 367.4515} C_DIS
LIN {X 12.7525,Y 139.4804,Z 169,A 85.6693,B 9.5967,C 0.0763,E1 9.6114,E2 365.7112} C_DIS
LIN {X 8.9314,Y 139.776,Z 169,A 87.2535,B 9.5967,C 0.0757,E1 9.607,E2 364.1255} C_DIS
LIN {X 4.2671,Y 139.9963,Z 169,A 89.1156,B 9.5967,C 0.0765,E1 9.6018,E2 362.2703} C_DIS
LIN {X 0.7445,Y 140.0589,Z 169,A 90.5651,B 9.5967,C 0.0764,E1 9.5978,E2 360.8204} C_DIS
LIN {X -3.6411,Y 140.0137,Z 169,A 92.3692,B 9.5967,C 0.0763,E1 9.5927,E2 359.0159} C_DIS
LIN {X -7.6981,Y 139.8506,Z 169,A 94.2938,B 9.5967,C 0.0711,E1 9.5873,E2 357.0588} C_DIS
LIN {X -11.1744,Y 139.6156,Z 169,A 95.3883,B 9.5967,C 0.0783,E1 9.5843,E2 356.007} C_DIS
LIN {X -14.9801,Y 139.2573,Z 169,A 97.0263,B 9.5967,C 0.0773,E1 9.5798,E2 354.3604} C_DIS
LIN {X -18.9299,Y 138.7775,Z 169,A 99.211,B 9.5967,C 0.0664,E1 9.5735,E2 352.1059} C_DIS
LIN {X -23.9695,Y 137.9961,Z 169,A 100.808,B 9.5967,C 0.0776,E1 9.5693,E2 350.5725} C_DIS
LIN {X -30.7934,Y 136.6341,Z 169,A 103.591,B 9.5967,C 0.0807,E1 9.5617,E2 347.7993} C_DIS
LIN {X -34.4427,Y 135.7595,Z 169,A 105.0564,B 9.5967,C 0.0832,E1 9.5578,E2 346.3437} C_DIS
LIN {X -37.6942,Y 134.8928,Z 169,A 106.5209,B 9.5967,C 0.0825,E1 9.5538,E2 344.8691} C_DIS
LIN {X -41.9246,Y 133.6404,Z 169,A 108.3912,B 9.5967,C 0.0828,E1 9.5488,E2 342.9918} C_DIS
LIN {X -44.8733,Y 132.679,Z 169,A 109.8011,B 9.5967,C 0.0812,E1 9.545,E2 341.565} C_DIS
LIN {X -50.3583,Y 130.6947,Z 169,A 112.4368,B 9.5967,C 0.0787,E1 9.538,E2 338.8995} C_DIS
LIN {X -54.4137,Y 129.0591,Z 169,A 113.7583,B 9.5966,C 0.0901,E1 9.5348,E2 337.6387} C_DIS
LIN {X -59.78,Y 126.6636,Z 169,A 116.2252,B 9.5966,C 0.0918,E1 9.5285,E2 335.1658} C_DIS
LIN {X -63.0497,Y 125.0676,Z 169,A 117.6661,B 9.5966,C 0.0947,E1 9.5249,E2 333.7322} C_DIS
LIN {X -66.6105,Y 123.2096,Z 169,A 119.2971,B 9.5966,C 0.0973,E1 9.5209,E2 332.1041} C_DIS
LIN {X -70.8255,Y 120.8354,Z 169,A 121.402,B 9.5966,C 0.0977,E1 9.5158,E2 329.9851} C_DIS
LIN {X -74.3882,Y 118.6761,Z 169,A 122.9332,B 9.5964,C 0.1038,E1 9.5122,E2 328.4773} C_DIS
LIN {X -77.3028,Y 116.7982,Z 169,A 124.581,B 9.5964,C 0.1016,E1 9.5083,E2 326.8018} C_DIS
LIN {X -81.1278,Y 114.1747,Z 169,A 126.2222,B 9.5964,C 0.1098,E1 9.5046,E2 325.1947} C_DIS
LIN {X -85.3965,Y 111.018,Z 169,A 129.1681,B 9.5964,C 0.0987,E1 9.4978,E2 322.1528} C_DIS
LIN {X -89.228,Y 107.9621,Z 169,A 130.6785,B 9.5964,C 0.112,E1 9.4947,E2 320.7071} C_DIS
LIN {X -91.8629,Y 105.7295,Z 169,A 131.9809,B 9.5963,C 0.1168,E1 9.492,E2 319.42} C_DIS
LIN {X -95.1454,Y 102.7859,Z 169,A 134.7234,B 9.5965,C 0.1025,E1 9.4861,E2 316.5599} C_DIS
LIN {X -99.7681,Y 98.3049,Z 169,A 136.6321,B 9.5962,C 0.1218,E1 9.4825,E2 314.7464} C_DIS
LIN {X -106.3186,Y 91.1804,Z 169,A 140.6049,B 9.5962,C 0.1303,E1 9.4751,E2 310.7761} C_DIS
LIN {X -109.0788,Y 87.8592,Z 169,A 142.4821,B 9.5961,C 0.1323,E1 9.4717,E2 308.8866} C_DIS
LIN {X -111.981,Y 84.1295,Z 169,A 144.3615,B 9.5961,C 0.1378,E1 9.4686,E2 307.0161} C_DIS
LIN {X -114.6352,Y 80.4755,Z 169,A 146.2531,B 9.596,C 0.1414,E1 9.4655,E2 305.1209} C_DIS
LIN {X -117.441,Y 76.322,Z 169,A 148.9402,B 9.596,C 0.1346,E1 9.4613,E2 302.3547} C_DIS
LIN {X -120.4179,Y 71.5333,Z 169,A 150.4658,B 9.5958,C 0.1549,E1 9.4592,E2 300.9312} C_DIS
LIN {X -122.3128,Y 68.2437,Z 169,A 152.2457,B 9.5958,C 0.1547,E1 9.4567,E2 299.1242} C_DIS
LIN {X -124.4949,Y 64.1747,Z 169,A 154.0794,B 9.5957,C 0.1606,E1 9.4543,E2 297.2995} C_DIS
LIN {X -126.1969,Y 60.7568,Z 169,A 155.6398,B 9.5956,C 0.1648,E1 9.4524,E2 295.7409} C_DIS
LIN {X -127.5676,Y 57.8262,Z 169,A 157.1412,B 9.5956,C 0.165,E1 9.4507,E2 294.2183} C_DIS
LIN {X -129.2208,Y 54.0265,Z 169,A 158.6254,B 9.5954,C 0.1735,E1 9.4491,E2 292.7627} C_DIS
LIN {X -130.8067,Y 50.0703,Z 169,A 160.595,B 9.5954,C 0.1741,E1 9.447,E2 290.7663} C_DIS
LIN {X -132.2581,Y 46.0951,Z 169,A 162.262,B 9.5954,C 0.1801,E1 9.4455,E2 289.1092} C_DIS
LIN {X -133.3936,Y 42.6974,Z 169,A 163.4978,B 9.5952,C 0.1883,E1 9.4444,E2 287.9042} C_DIS
LIN {X -134.3523,Y 39.578,Z 169,A 165.1052,B 9.5952,C 0.1871,E1 9.4431,E2 286.2636} C_DIS
LIN {X -135.2487,Y 36.3979,Z 169,A 166.471,B 9.5952,C 0.1907,E1 9.4421,E2 284.8974} C_DIS
LIN {X -136.1815,Y 32.7346,Z 169,A 167.9899,B 9.595,C 0.1956,E1 9.4411,E2 283.3836} C_DIS
LIN {X -136.944,Y 29.3822,Z 169,A 169.4785,B 9.595,C 0.1981,E1 9.4402,E2 281.886} C_DIS
LIN {X -137.7654,Y 25.2588,Z 169,A 171.2311,B 9.5949,C 0.2024,E1 9.4393,E2 280.131} C_DIS
LIN {X -138.3946,Y 21.5387,Z 169,A 172.7536,B 9.5948,C 0.2073,E1 9.4386,E2 278.6128} C_DIS
LIN {X -138.8926,Y 18.0515,Z 169,A 174.2443,B 9.5948,C 0.2105,E1 9.438,E2 277.1172} C_DIS
LIN {X -139.2345,Y 15.192,Z 169,A 175.9393,B 9.5948,C 0.2045,E1 9.4375,E2 275.3572} C_DIS
LIN {X -139.6602,Y 10.5913,Z 169,A 177.2589,B 9.5945,C 0.2204,E1 9.4372,E2 274.1126} C_DIS
LIN {X -139.9891,Y 4.5255,Z 169,A 179.8386,B 9.5944,C 0.226,E1 9.4369,E2 271.5234} C_DIS
LIN {X -140.0149,Y -3.5988,Z 169,A -175.9331,B 9.5945,C 0.219,E1 9.4369,E2 267.1818} C_DIS
LIN {X -139.7141,Y -9.8538,Z 169,A -174.2132,B 9.594,C 0.242,E1 9.4373,E2 265.573} C_DIS
LIN {X -139.1994,Y -15.5182,Z 169,A -171.7049,B 9.5939,C 0.2454,E1 9.438,E2 263.0436} C_DIS
LIN {X -138.7363,Y -19.2238,Z 169,A -170.2869,B 9.5937,C 0.2518,E1 9.4385,E2 261.641} C_DIS
LIN {X -138.184,Y -22.8514,Z 169,A -168.7216,B 9.5937,C 0.2549,E1 9.4392,E2 260.0687} C_DIS
LIN {X -137.5799,Y -26.2435,Z 169,A -167.3502,B 9.5935,C 0.2596,E1 9.4399,E2 258.7034} C_DIS
LIN {X -136.9088,Y -29.5452,Z 169,A -165.8955,B 9.5935,C 0.2621,E1 9.4407,E2 257.2401} C_DIS
LIN {X -136.1899,Y -32.6994,Z 169,A -164.5644,B 9.5934,C 0.2657,E1 9.4415,E2 255.9091} C_DIS
LIN {X -135.3689,Y -35.9473,Z 169,A -163.2276,B 9.5932,C 0.2701,E1 9.4425,E2 254.5777} C_DIS
LIN {X -134.2652,Y -39.8757,Z 169,A -161.4543,B 9.5932,C 0.2729,E1 9.4438,E2 252.7925} C_DIS
LIN {X -132.9851,Y -43.954,Z 169,A -159.6896,B 9.593,C 0.2774,E1 9.4454,E2 251.027} C_DIS
LIN {X -132.0154,Y -46.791,Z 169,A -158.3527,B 9.593,C 0.2787,E1 9.4466,E2 249.6769} C_DIS
LIN {X -130.8523,Y -49.9514,Z 169,A -157.0753,B 9.5928,C 0.2842,E1 9.4478,E2 248.4135} C_DIS
LIN {X -129.4344,Y -53.515,Z 169,A -155.3945,B 9.5928,C 0.2863,E1 9.4496,E2 246.7193} C_DIS
LIN {X -127.9117,Y -57.0569,Z 169,A -153.8757,B 9.5926,C 0.2915,E1 9.4513,E2 245.2091} C_DIS
LIN {X -126.5345,Y -60.0502,Z 169,A -152.4805,B 9.5926,C 0.2942,E1 9.453,E2 243.8087} C_DIS
LIN {X -124.9653,Y -63.2507,Z 169,A -151.0321,B 9.5924,C 0.2981,E1 9.4548,E2 242.3625} C_DIS
LIN {X -123.0523,Y -66.8998,Z 169,A -149.198,B 9.5924,C 0.2995,E1 9.4572,E2 240.5103} C_DIS
LIN {X -120.7223,Y -71.0181,Z 169,A -147.2549,B 9.5922,C 0.3042,E1 9.4599,E2 238.5674} C_DIS
LIN {X -118.2843,Y -75.009,Z 169,A -145.321,B 9.5921,C 0.3084,E1 9.4628,E2 236.6319} C_DIS
LIN {X -115.8121,Y -78.7724,Z 169,A -143.4927,B 9.5919,C 0.313,E1 9.4656,E2 234.8064} C_DIS
LIN {X -113.298,Y -82.347,Z 169,A -141.2069,B 9.5921,C 0.3076,E1 9.4695,E2 232.4567} C_DIS
LIN {X -110.4324,Y -86.1528,Z 169,A -139.6211,B 9.5917,C 0.319,E1 9.4721,E2 230.9192} C_DIS
LIN {X -107.1685,Y -90.1797,Z 169,A -136.6663,B 9.5921,C 0.3073,E1 9.4776,E2 227.8561} C_DIS
LIN {X -102.603,Y -95.3418,Z 169,A -134.6603,B 9.5914,C 0.3291,E1 9.4812,E2 225.9579} C_DIS
LIN {X -100.2561,Y -97.8074,Z 169,A -133.1643,B 9.5914,C 0.3299,E1 9.4841,E2 224.4489} C_DIS
LIN {X -96.6218,Y -101.3987,Z 169,A -131.1543,B 9.5912,C 0.3355,E1 9.4881,E2 222.4501} C_DIS
LIN {X -93.2621,Y -104.4972,Z 169,A -129.1026,B 9.5912,C 0.3355,E1 9.4924,E2 220.3751} C_DIS
LIN {X -89.4959,Y -107.7402,Z 169,A -127.1847,B 9.591,C 0.3413,E1 9.4965,E2 218.4729} C_DIS
LIN {X -85.5928,Y -110.8664,Z 169,A -124.306,B 9.5914,C 0.3281,E1 9.5031,E2 215.4851} C_DIS
LIN {X -80.1025,Y -114.8957,Z 169,A -122.3315,B 9.5907,C 0.3489,E1 9.5073,E2 213.618} C_DIS
LIN {X -76.2364,Y -117.4966,Z 169,A -120.4484,B 9.5906,C 0.3523,E1 9.5117,E2 211.7382} C_DIS
LIN {X -72.723,Y -119.7033,Z 169,A -118.7009,B 9.5906,C 0.3537,E1 9.5159,E2 209.9843} C_DIS
LIN {X -68.8826,Y -121.9537,Z 169,A -115.72,B 9.5913,C 0.3323,E1 9.5235,E2 206.8503} C_DIS
LIN {X -61.349,Y -125.9112,Z 169,A -113.4053,B 9.5903,C 0.3606,E1 9.5289,E2 204.69} C_DIS
LIN {X -56.5884,Y -128.1213,Z 169,A -111.2888,B 9.5902,C 0.3636,E1 9.5343,E2 202.5775} C_DIS
LIN {X -52.7307,Y -129.7556,Z 169,A -109.6522,B 9.59,C 0.3669,E1 9.5384,E2 200.9509} C_DIS
LIN {X -49.8338,Y -130.8971,Z 169,A -108.1674,B 9.5902,C 0.3637,E1 9.5424,E2 199.4384} C_DIS
LIN {X -45.995,Y -132.2928,Z 169,A -106.6393,B 9.59,C 0.3681,E1 9.5464,E2 197.9287} C_DIS
LIN {X -42.6889,Y -133.3963,Z 169,A -105.1664,B 9.59,C 0.3683,E1 9.5503,E2 196.4495} C_DIS
LIN {X -39.3747,Y -134.4119,Z 169,A -103.9587,B 9.5898,C 0.3737,E1 9.5534,E2 195.269} C_DIS
LIN {X -33.963,Y -135.8812,Z 169,A -101.4032,B 9.5899,C 0.3697,E1 9.5604,E2 192.6789} C_DIS
LIN {X -29.9558,Y -136.8202,Z 169,A -99.6793,B 9.5899,C 0.3697,E1 9.5651,E2 190.9493} C_DIS
LIN {X -26.4885,Y -137.5331,Z 169,A -98.1387,B 9.5899,C 0.3683,E1 9.5694,E2 189.3962} C_DIS
LIN {X -21.702,Y -138.3693,Z 169,A -96.4683,B 9.5897,C 0.3758,E1 9.5739,E2 187.7668} C_DIS
LIN {X -19.0231,Y -138.7644,Z 169,A -95.0916,B 9.5899,C 0.3704,E1 9.5778,E2 186.3545} C_DIS
LIN {X -15.7595,Y -139.1734,Z 169,A -93.7376,B 9.5899,C 0.3704,E1 9.5816,E2 184.9989} C_DIS
LIN {X -12.2336,Y -139.5261,Z 169,A -92.52,B 9.5897,C 0.3757,E1 9.5849,E2 183.8112} C_DIS
LIN {X -8.9381,Y -139.7756,Z 169,A -90.9831,B 9.5899,C 0.3718,E1 9.5892,E2 182.2494} C_DIS
LIN {X -4.8076,Y -139.9798,Z 169,A -89.2429,B 9.5899,C 0.3707,E1 9.5941,E2 180.5022} C_DIS
LIN {X -0.6128,Y -140.0596,Z 169,A -87.634,B 9.5899,C 0.3729,E1 9.5985,E2 178.9066} C_DIS
LIN {X -0.6128,Y -140.0596,Z 169,A -87.634,B 9.5899,C 0.3729,E1 9.5985,E2 178.9066} C_DIS
Enddeposition()
LIN {X 1.0246,Y -140.9657,Z 169,A -87.1642,B 9.5896,C 0.3829,E1 9.5998,E2 178.4966} C_DIS
Startdeposition()
$VEL.CP = VEL_PRINT
LIN {X -1.726,Y -140.964,Z 169,A -88.7127,B 9.5892,C 0.3925,E1 9.5953,E2 180.1025} C_DIS
LIN {X -5.179,Y -140.8783,Z 169,A -90.1106,B 9.5892,C 0.3925,E1 9.5914,E2 181.5003} C_DIS
LIN {X -8.6292,Y -140.7087,Z 169,A -91.5717,B 9.5892,C 0.3936,E1 9.5873,E2 182.9694} C_DIS
LIN {X -12.768,Y -140.3954,Z 169,A -93.3028,B 9.5892,C 0.3944,E1 9.5825,E2 184.7069} C_DIS
LIN {X -16.5822,Y -139.9944,Z 169,A -94.8466,B 9.5892,C 0.3937,E1 9.5782,E2 186.2493} C_DIS
LIN {X -20.6752,Y -139.4506,Z 169,A -96.4273,B 9.5892,C 0.3912,E1 9.5739,E2 187.8179} C_DIS
LIN {X -24.0946,Y -138.9006,Z 169,A -97.8063,B 9.5892,C 0.39,E1 9.5701,E2 189.1935} C_DIS
LIN {X -26.8421,Y -138.3944,Z 169,A -98.9801,B 9.5892,C 0.3904,E1 9.5669,E2 190.3727} C_DIS
LIN {X -30.875,Y -137.5513,Z 169,A -100.8042,B 9.5892,C 0.3927,E1 9.5618,E2 192.2167} C_DIS
LIN {X -35.26,Y -136.4933,Z 169,A -102.4997,B 9.5893,C 0.3887,E1 9.5573,E2 193.8947} C_DIS
LIN {X -38.5954,Y -135.5881,Z 169,A -103.8815,B 9.5893,C 0.3873,E1 9.5536,E2 195.2738} C_DIS
LIN {X -41.9307,Y -134.5943,Z 169,A -105.3166,B 9.5894,C 0.3867,E1 9.5497,E2 196.7119} C_DIS
LIN {X -45.2231,Y -133.5242,Z 169,A -106.8678,B 9.5894,C 0.3886,E1 9.5456,E2 198.282} C_DIS
LIN {X -49.7482,Y -131.9034,Z 169,A -108.7099,B 9.5895,C 0.3846,E1 9.5408,E2 200.1098} C_DIS
LIN {X -53.3204,Y -130.5016,Z 169,A -110.2801,B 9.5895,C 0.3833,E1 9.5367,E2 201.6815} C_DIS
LIN {X -56.5047,Y -129.1544,Z 169,A -111.6811,B 9.5896,C 0.3817,E1 9.5331,E2 203.0821} C_DIS
LIN {X -59.4949,Y -127.8036,Z 169,A -113.0327,B 9.5896,C 0.3806,E1 9.5297,E2 204.436} C_DIS
LIN {X -62.59,Y -126.3163,Z 169,A -114.4761,B 9.5896,C 0.38,E1 9.526,E2 205.8856} C_DIS
LIN {X -66.4247,Y -124.3451,Z 169,A -116.302,B 9.5897,C 0.3793,E1 9.5215,E2 207.7212} C_DIS
LIN {X -70.2359,Y -122.2332,Z 169,A -118.0571,B 9.5898,C 0.3766,E1 9.5172,E2 209.4741} C_DIS
LIN {X -73.9528,Y -120.0204,Z 169,A -119.8105,B 9.5899,C 0.3741,E1 9.513,E2 211.2267} C_DIS
LIN {X -77.5946,Y -117.6984,Z 169,A -121.6036,B 9.5899,C 0.3722,E1 9.5088,E2 213.0245} C_DIS
LIN {X -81.11,Y -115.3041,Z 169,A -123.3577,B 9.5901,C 0.37,E1 9.5048,E2 214.7815} C_DIS
LIN {X -84.5908,Y -112.7759,Z 169,A -125.1052,B 9.5901,C 0.3671,E1 9.5009,E2 216.5286} C_DIS
LIN {X -88.0876,Y -110.0661,Z 169,A -126.9116,B 9.5903,C 0.3642,E1 9.4969,E2 218.3356} C_DIS
LIN {X -91.4194,Y -107.3143,Z 169,A -128.7056,B 9.5903,C 0.3618,E1 9.493,E2 220.1341} C_DIS
LIN {X -94.6723,Y -104.4557,Z 169,A -130.4819,B 9.5905,C 0.3589,E1 9.4893,E2 221.912} C_DIS
LIN {X -97.8303,Y -101.5045,Z 169,A -132.2734,B 9.5905,C 0.3562,E1 9.4857,E2 223.7074} C_DIS
LIN {X -100.9024,Y -98.4513,Z 169,A -134.0126,B 9.5907,C 0.3523,E1 9.4823,E2 225.4433} C_DIS
LIN {X -103.8596,Y -95.3259,Z 169,A -135.769,B 9.5909,C 0.3488,E1 9.4789,E2 227.2} C_DIS
LIN {X -106.7238,Y -92.108,Z 169,A -137.5845,B 9.5909,C 0.3464,E1 9.4756,E2 229.0231} C_DIS
LIN {X -109.5212,Y -88.764,Z 169,A -139.3867,B 9.5911,C 0.3431,E1 9.4724,E2 230.8284} C_DIS
LIN {X -112.1855,Y -85.372,Z 169,A -141.1159,B 9.5912,C 0.3387,E1 9.4694,E2 232.5537} C_DIS
LIN {X -114.7584,Y -81.8802,Z 169,A -142.8894,B 9.5914,C 0.3349,E1 9.4665,E2 234.3276} C_DIS
LIN {X -117.2133,Y -78.3254,Z 169,A -144.7027,B 9.5914,C 0.3318,E1 9.4637,E2 236.1474} C_DIS
LIN {X -119.5588,Y -74.6967,Z 169,A -146.4675,B 9.5916,C 0.3278,E1 9.461,E2 237.9123} C_DIS
LIN {X -121.8007,Y -70.983,Z 169,A -148.2924,B 9.5917,C 0.3246,E1 9.4584,E2 239.7442} C_DIS
LIN {X -123.9164,Y -67.221,Z 169,A -150.0793,B 9.5918,C 0.3208,E1 9.456,E2 241.5342} C_DIS
LIN {X -125.7684,Y -63.6841,Z 169,A -151.6447,B 9.592,C 0.3156,E1 9.454,E2 243.0911} C_DIS
LIN {X -127.437,Y -60.2775,Z 169,A -153.1739,B 9.5921,C 0.3114,E1 9.4522,E2 244.6176} C_DIS
LIN {X -128.7619,Y -57.3907,Z 169,A -154.5171,B 9.5922,C 0.309,E1 9.4506,E2 245.9667} C_DIS
LIN {X -130.4181,Y -53.527,Z 169,A -156.3741,B 9.5922,C 0.3072,E1 9.4486,E2 247.8416} C_DIS
LIN {X -131.906,Y -49.7413,Z 169,A -157.8874,B 9.5925,C 0.3002,E1 9.4471,E2 249.3356} C_DIS
LIN {X -133.3065,Y -45.8563,Z 169,A -159.5915,B 9.5926,C 0.2961,E1 9.4455,E2 251.0418} C_DIS
LIN {X -134.3893,Y -42.5787,Z 169,A -161.0142,B 9.5927,C 0.2926,E1 9.4443,E2 252.4659} C_DIS
LIN {X -135.3917,Y -39.2752,Z 169,A -162.4379,B 9.5928,C 0.2891,E1 9.4431,E2 253.8911} C_DIS
LIN {X -136.4887,Y -35.278,Z 169,A -164.2495,B 9.5928,C 0.2868,E1 9.4418,E2 255.7177} C_DIS
LIN {X -137.3983,Y -31.545,Z 169,A -165.736,B 9.5931,C 0.281,E1 9.4409,E2 257.1932} C_DIS
LIN {X -138.2649,Y -27.5054,Z 169,A -167.4316,B 9.5931,C 0.2766,E1 9.4399,E2 258.8896} C_DIS
LIN {X -138.8985,Y -24.1061,Z 169,A -168.8564,B 9.5933,C 0.2729,E1 9.4392,E2 260.3156} C_DIS
LIN {X -139.4495,Y -20.6828,Z 169,A -170.3112,B 9.5933,C 0.2697,E1 9.4386,E2 261.775} C_DIS
LIN {X -139.914,Y -17.2562,Z 169,A -171.8745,B 9.5934,C 0.2685,E1 9.438,E2 263.3572} C_DIS
LIN {X -140.3967,Y -12.7543,Z 169,A -173.574,B 9.5936,C 0.2607,E1 9.4375,E2 265.0371} C_DIS
LIN {X -140.6657,Y -9.3272,Z 169,A -174.9389,B 9.5938,C 0.256,E1 9.4373,E2 266.3965} C_DIS
LIN {X -140.8359,Y -6.2656,Z 169,A -176.2979,B 9.5938,C 0.2545,E1 9.4371,E2 267.7688} C_DIS
LIN {X -140.9518,Y -2.4591,Z 169,A -177.8896,B 9.5938,C 0.2507,E1 9.437,E2 269.3646} C_DIS
LIN {X -140.9537,Y 2.3453,Z 169,A -179.8856,B 9.594,C 0.2458,E1 9.437,E2 271.3642} C_DIS
LIN {X -140.8374,Y 6.2277,Z 169,A 178.5593,B 9.5941,C 0.2408,E1 9.4372,E2 272.9149} C_DIS
LIN {X -140.6682,Y 9.2873,Z 169,A 177.3144,B 9.5942,C 0.2372,E1 9.4374,E2 274.1585} C_DIS
LIN {X -140.3987,Y 12.7339,Z 169,A 175.7604,B 9.5942,C 0.2358,E1 9.4377,E2 275.73} C_DIS
LIN {X -139.9141,Y 17.2555,Z 169,A 174.0031,B 9.5944,C 0.2288,E1 9.4383,E2 277.4738} C_DIS
LIN {X -139.4484,Y 20.6906,Z 169,A 172.5689,B 9.5945,C 0.2252,E1 9.4388,E2 278.9098} C_DIS
LIN {X -138.8989,Y 24.1039,Z 169,A 171.1785,B 9.5946,C 0.2209,E1 9.4395,E2 280.2969} C_DIS
LIN {X -138.3947,Y 26.8406,Z 169,A 169.8745,B 9.5946,C 0.2207,E1 9.4402,E2 281.6216} C_DIS
LIN {X -137.3988,Y 31.5426,Z 169,A 168.0016,B 9.5948,C 0.2137,E1 9.4413,E2 283.4823} C_DIS
LIN {X -136.4876,Y 35.2826,Z 169,A 166.4162,B 9.5948,C 0.2096,E1 9.4424,E2 285.0688} C_DIS
LIN {X -135.5817,Y 38.6185,Z 169,A 164.9888,B 9.595,C 0.2061,E1 9.4434,E2 286.4976} C_DIS
Enddeposition()
END
